      A     M   2002.5;
      =     L      0.0;
      BLD   103;
      A     I    367.3;
      =     L      0.1;
      BLD   103;
      A     I    367.4;
      =     L      0.2;
      BLD   103;
      A     I    367.6;
      =     L      0.4;
      BLD   103;
      A     I    367.7;
      =     L      0.6;
      BLD   103;
      A     I    368.0;
      =     L      1.0;
      BLD   103;
      A     I    368.1;
      =     L      1.2;
      BLD   103;
      A     M   2241.6;
      =     L      2.1;
      BLD   103;
      A     M   2241.7;
      =     L      2.2;
      BLD   103;
      AN    M   2004.0;
      AN    M   2004.1;
      AN    M   6060.1;
      AN    M   6460.0;
      AN    M   6480.0;
      AN    M   2004.2;
      A     M   2000.2;
      =     L      2.3;
      BLD   103;
      A(    ;
      O     I    150.1;
      O     I      0.1;
      )     ;
      =     L      2.5;
      BLD   103;
      A     M      0.5;
      =     L      2.6;
      BLD   103;
      CALL #S704_TL_DC_2ND_CLAMP2 (
           Enable_Aux               := L      0.0,
           Adv_Amount               := 1,
           Ret_Amount               := 5,
           LS_Adv1                  := L      0.1,
           LS_Ret1                  := L      0.2,
           LS_Ret2                  := L      0.4,
           LS_Ret3                  := L      0.6,
           LS_Ret4                  := L      1.0,
           LS_Ret5                  := L      1.2,
           SOL_Adv                  := L      2.1,
           SOL_Ret                  := L      2.2,
           M_Ready                  := L      2.3,
           T_CHK1                   := T#4S,
           T_CHK2                   := T#4S,
           PB_Error_Rst             := L      2.5,
           M_FLICK                  := L      2.6,
           M_Adv_Err                := M   2251.6,
           M_Ret_Err                := M   2251.7,
           Visu_Adv                 := DB51.DBW  748,
           Visu_Ret                 := DB51.DBW  750);
      NOP   0;
NETWORK
TITLE =
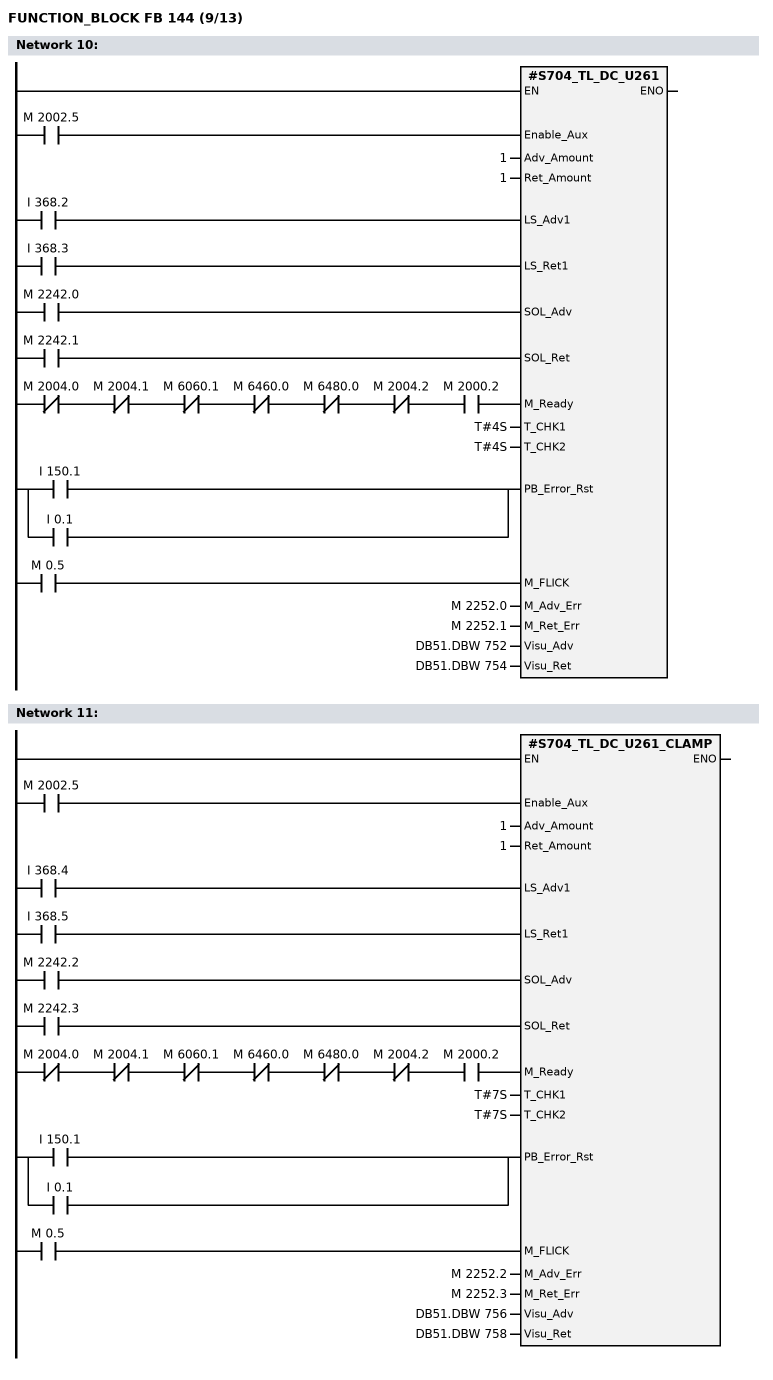

      A     M   2002.5;
      =     L      0.0;
      BLD   103;
      A     I    368.2;
      =     L      0.1;
      BLD   103;
      A     I    368.3;
      =     L      0.2;
      BLD   103;
      A     M   2242.0;
      =     L      2.1;
      BLD   103;
      A     M   2242.1;
      =     L      2.2;
      BLD   103;
      AN    M   2004.0;
      AN    M   2004.1;
      AN    M   6060.1;
      AN    M   6460.0;
      AN    M   6480.0;
      AN    M   2004.2;
      A     M   2000.2;
      =     L      2.3;
      BLD   103;
      A(    ;
      O     I    150.1;
      O     I      0.1;
      )     ;
      =     L      2.5;
      BLD   103;
      A     M      0.5;
      =     L      2.6;
      BLD   103;
      CALL #S704_TL_DC_U261 (
           Enable_Aux               := L      0.0,
           Adv_Amount               := 1,
           Ret_Amount               := 1,
           LS_Adv1                  := L      0.1,
           LS_Ret1                  := L      0.2,
           SOL_Adv                  := L      2.1,
           SOL_Ret                  := L      2.2,
           M_Ready                  := L      2.3,
           T_CHK1                   := T#4S,
           T_CHK2                   := T#4S,
           PB_Error_Rst             := L      2.5,
           M_FLICK                  := L      2.6,
           M_Adv_Err                := M   2252.0,
           M_Ret_Err                := M   2252.1,
           Visu_Adv                 := DB51.DBW  752,
           Visu_Ret                 := DB51.DBW  754);
      NOP   0;
NETWORK
TITLE =

      A     M   2002.5;
      =     L      0.0;
      BLD   103;
      A     I    368.4;
      =     L      0.1;
      BLD   103;
      A     I    368.5;
      =     L      0.2;
      BLD   103;
      A     M   2242.2;
      =     L      2.1;
      BLD   103;
      A     M   2242.3;
      =     L      2.2;
      BLD   103;
      AN    M   2004.0;
      AN    M   2004.1;
      AN    M   6060.1;
      AN    M   6460.0;
      AN    M   6480.0;
      AN    M   2004.2;
      A     M   2000.2;
      =     L      2.3;
      BLD   103;
      A(    ;
      O     I    150.1;
      O     I      0.1;
      )     ;
      =     L      2.5;
      BLD   103;
      A     M      0.5;
      =     L      2.6;
      BLD   103;
      CALL #S704_TL_DC_U261_CLAMP (
           Enable_Aux               := L      0.0,
           Adv_Amount               := 1,
           Ret_Amount               := 1,
           LS_Adv1                  := L      0.1,
           LS_Ret1                  := L      0.2,
           SOL_Adv                  := L      2.1,
           SOL_Ret                  := L      2.2,
           M_Ready                  := L      2.3,
           T_CHK1                   := T#7S,
           T_CHK2                   := T#7S,
           PB_Error_Rst             := L      2.5,
           M_FLICK                  := L      2.6,
           M_Adv_Err                := M   2252.2,
           M_Ret_Err                := M   2252.3,
           Visu_Adv                 := DB51.DBW  756,
           Visu_Ret                 := DB51.DBW  758);
      NOP   0;
NETWORK
TITLE =
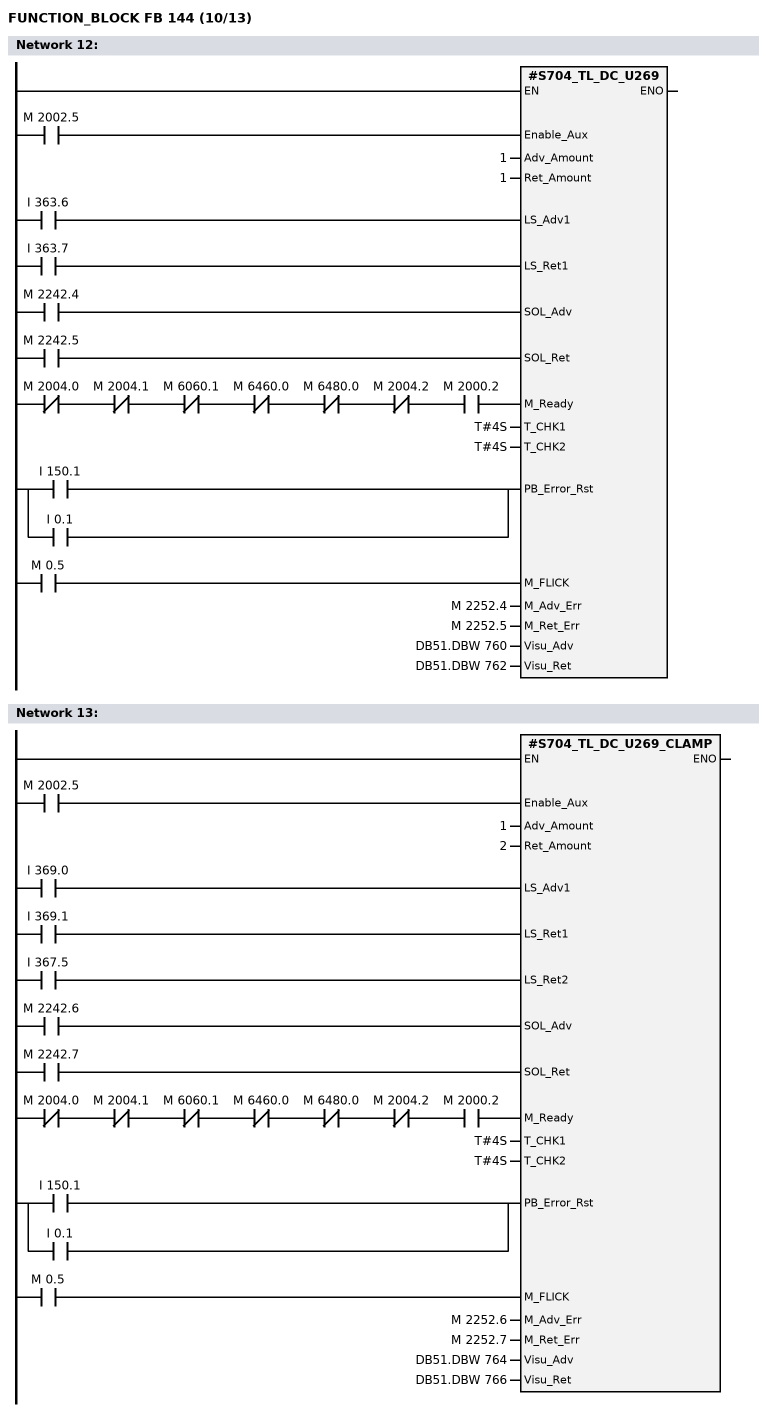

      A     M   2002.5;
      =     L      0.0;
      BLD   103;
      A     I    363.6;
      =     L      0.1;
      BLD   103;
      A     I    363.7;
      =     L      0.2;
      BLD   103;
      A     M   2242.4;
      =     L      2.1;
      BLD   103;
      A     M   2242.5;
      =     L      2.2;
      BLD   103;
      AN    M   2004.0;
      AN    M   2004.1;
      AN    M   6060.1;
      AN    M   6460.0;
      AN    M   6480.0;
      AN    M   2004.2;
      A     M   2000.2;
      =     L      2.3;
      BLD   103;
      A(    ;
      O     I    150.1;
      O     I      0.1;
      )     ;
      =     L      2.5;
      BLD   103;
      A     M      0.5;
      =     L      2.6;
      BLD   103;
      CALL #S704_TL_DC_U269 (
           Enable_Aux               := L      0.0,
           Adv_Amount               := 1,
           Ret_Amount               := 1,
           LS_Adv1                  := L      0.1,
           LS_Ret1                  := L      0.2,
           SOL_Adv                  := L      2.1,
           SOL_Ret                  := L      2.2,
           M_Ready                  := L      2.3,
           T_CHK1                   := T#4S,
           T_CHK2                   := T#4S,
           PB_Error_Rst             := L      2.5,
           M_FLICK                  := L      2.6,
           M_Adv_Err                := M   2252.4,
           M_Ret_Err                := M   2252.5,
           Visu_Adv                 := DB51.DBW  760,
           Visu_Ret                 := DB51.DBW  762);
      NOP   0;
NETWORK
TITLE =

      A     M   2002.5;
      =     L      0.0;
      BLD   103;
      A     I    369.0;
      =     L      0.1;
      BLD   103;
      A     I    369.1;
      =     L      0.2;
      BLD   103;
      A     I    367.5;
      =     L      0.4;
      BLD   103;
      A     M   2242.6;
      =     L      2.1;
      BLD   103;
      A     M   2242.7;
      =     L      2.2;
      BLD   103;
      AN    M   2004.0;
      AN    M   2004.1;
      AN    M   6060.1;
      AN    M   6460.0;
      AN    M   6480.0;
      AN    M   2004.2;
      A     M   2000.2;
      =     L      2.3;
      BLD   103;
      A(    ;
      O     I    150.1;
      O     I      0.1;
      )     ;
      =     L      2.5;
      BLD   103;
      A     M      0.5;
      =     L      2.6;
      BLD   103;
      CALL #S704_TL_DC_U269_CLAMP (
           Enable_Aux               := L      0.0,
           Adv_Amount               := 1,
           Ret_Amount               := 2,
           LS_Adv1                  := L      0.1,
           LS_Ret1                  := L      0.2,
           LS_Ret2                  := L      0.4,
           SOL_Adv                  := L      2.1,
           SOL_Ret                  := L      2.2,
           M_Ready                  := L      2.3,
           T_CHK1                   := T#4S,
           T_CHK2                   := T#4S,
           PB_Error_Rst             := L      2.5,
           M_FLICK                  := L      2.6,
           M_Adv_Err                := M   2252.6,
           M_Ret_Err                := M   2252.7,
           Visu_Adv                 := DB51.DBW  764,
           Visu_Ret                 := DB51.DBW  766);
      NOP   0;
NETWORK
TITLE =
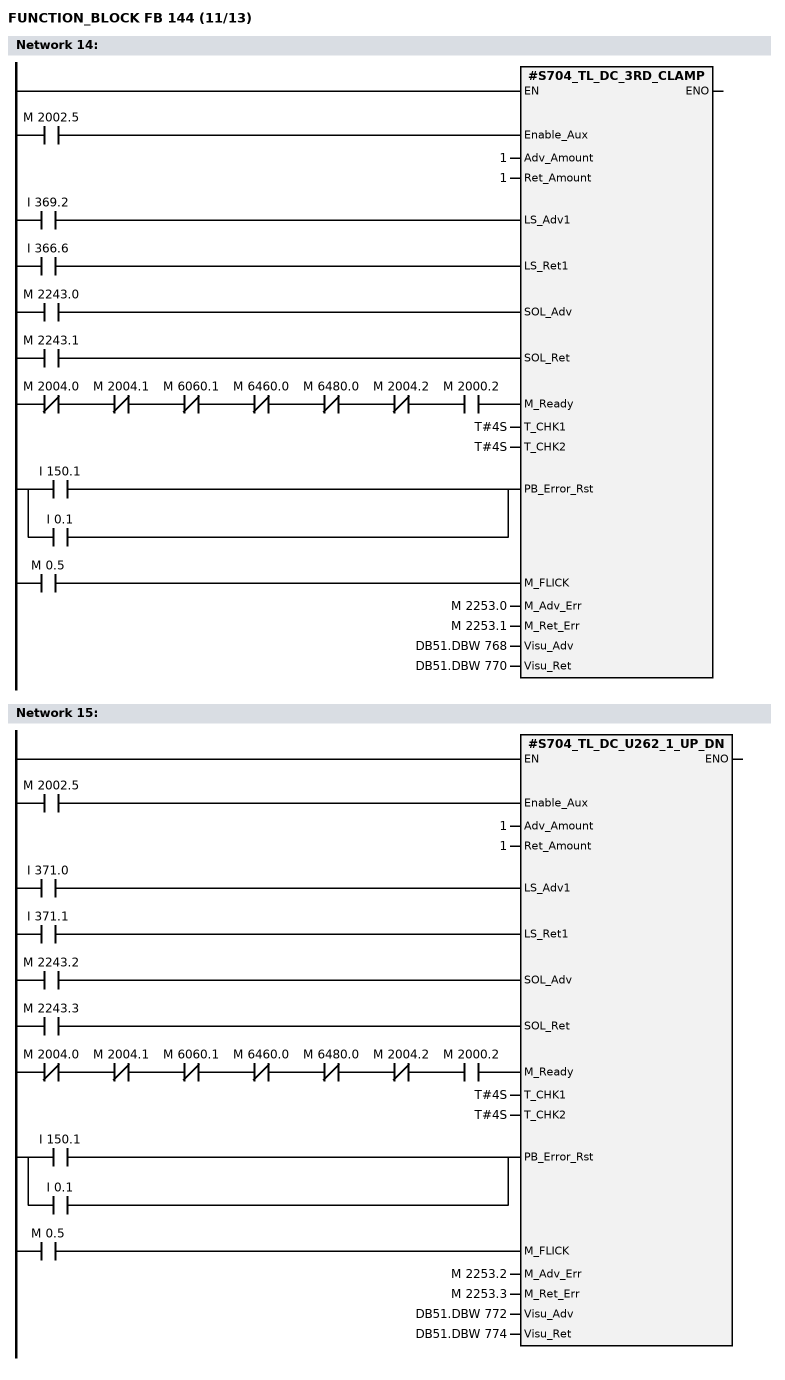

      A     M   2002.5;
      =     L      0.0;
      BLD   103;
      A     I    369.2;
      =     L      0.1;
      BLD   103;
      A     I    366.6;
      =     L      0.2;
      BLD   103;
      A     M   2243.0;
      =     L      2.1;
      BLD   103;
      A     M   2243.1;
      =     L      2.2;
      BLD   103;
      AN    M   2004.0;
      AN    M   2004.1;
      AN    M   6060.1;
      AN    M   6460.0;
      AN    M   6480.0;
      AN    M   2004.2;
      A     M   2000.2;
      =     L      2.3;
      BLD   103;
      A(    ;
      O     I    150.1;
      O     I      0.1;
      )     ;
      =     L      2.5;
      BLD   103;
      A     M      0.5;
      =     L      2.6;
      BLD   103;
      CALL #S704_TL_DC_3RD_CLAMP (
           Enable_Aux               := L      0.0,
           Adv_Amount               := 1,
           Ret_Amount               := 1,
           LS_Adv1                  := L      0.1,
           LS_Ret1                  := L      0.2,
           SOL_Adv                  := L      2.1,
           SOL_Ret                  := L      2.2,
           M_Ready                  := L      2.3,
           T_CHK1                   := T#4S,
           T_CHK2                   := T#4S,
           PB_Error_Rst             := L      2.5,
           M_FLICK                  := L      2.6,
           M_Adv_Err                := M   2253.0,
           M_Ret_Err                := M   2253.1,
           Visu_Adv                 := DB51.DBW  768,
           Visu_Ret                 := DB51.DBW  770);
      NOP   0;
NETWORK
TITLE =

      A     M   2002.5;
      =     L      0.0;
      BLD   103;
      A     I    371.0;
      =     L      0.1;
      BLD   103;
      A     I    371.1;
      =     L      0.2;
      BLD   103;
      A     M   2243.2;
      =     L      2.1;
      BLD   103;
      A     M   2243.3;
      =     L      2.2;
      BLD   103;
      AN    M   2004.0;
      AN    M   2004.1;
      AN    M   6060.1;
      AN    M   6460.0;
      AN    M   6480.0;
      AN    M   2004.2;
      A     M   2000.2;
      =     L      2.3;
      BLD   103;
      A(    ;
      O     I    150.1;
      O     I      0.1;
      )     ;
      =     L      2.5;
      BLD   103;
      A     M      0.5;
      =     L      2.6;
      BLD   103;
      CALL #S704_TL_DC_U262_1_UP_DN (
           Enable_Aux               := L      0.0,
           Adv_Amount               := 1,
           Ret_Amount               := 1,
           LS_Adv1                  := L      0.1,
           LS_Ret1                  := L      0.2,
           SOL_Adv                  := L      2.1,
           SOL_Ret                  := L      2.2,
           M_Ready                  := L      2.3,
           T_CHK1                   := T#4S,
           T_CHK2                   := T#4S,
           PB_Error_Rst             := L      2.5,
           M_FLICK                  := L      2.6,
           M_Adv_Err                := M   2253.2,
           M_Ret_Err                := M   2253.3,
           Visu_Adv                 := DB51.DBW  772,
           Visu_Ret                 := DB51.DBW  774);
      NOP   0;
NETWORK
TITLE =
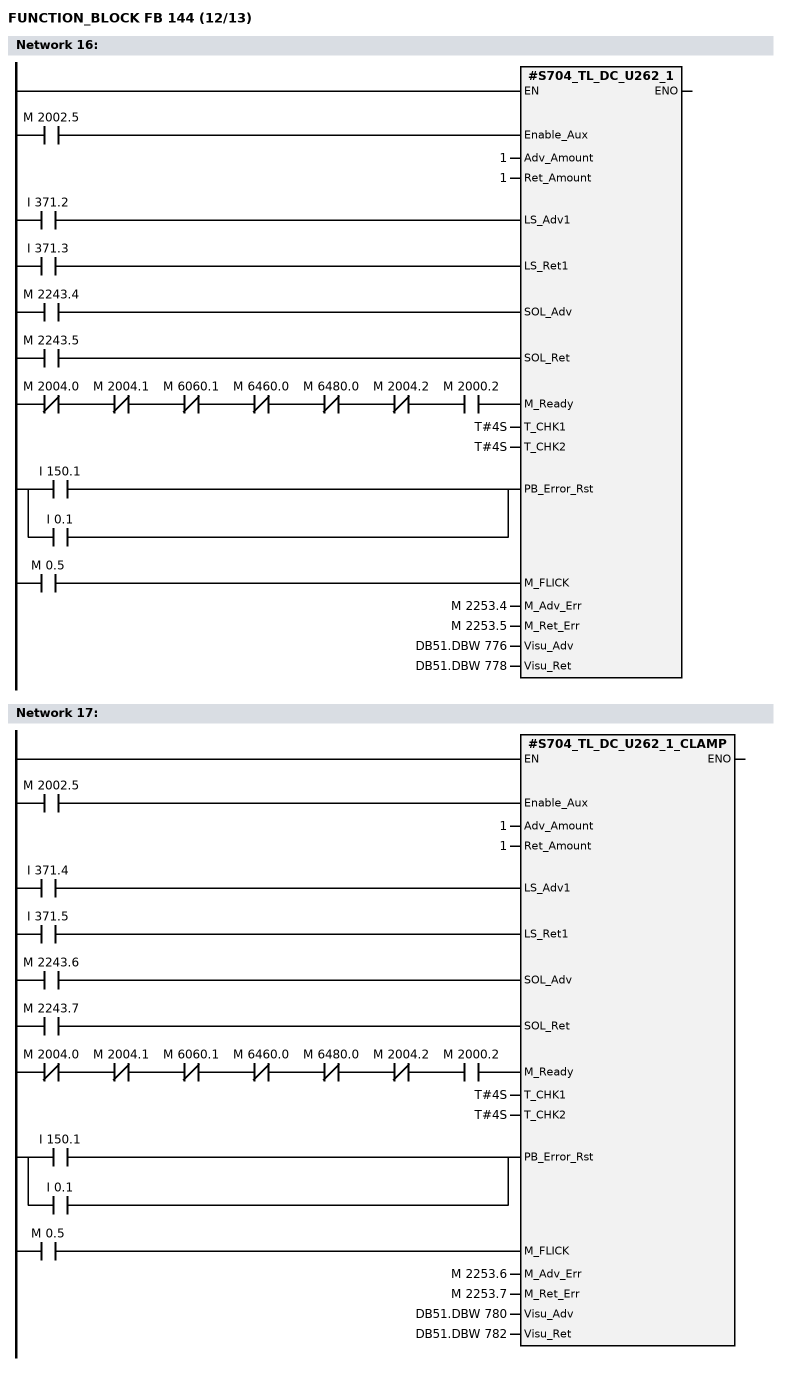

      A     M   2002.5;
      =     L      0.0;
      BLD   103;
      A     I    371.2;
      =     L      0.1;
      BLD   103;
      A     I    371.3;
      =     L      0.2;
      BLD   103;
      A     M   2243.4;
      =     L      2.1;
      BLD   103;
      A     M   2243.5;
      =     L      2.2;
      BLD   103;
      AN    M   2004.0;
      AN    M   2004.1;
      AN    M   6060.1;
      AN    M   6460.0;
      AN    M   6480.0;
      AN    M   2004.2;
      A     M   2000.2;
      =     L      2.3;
      BLD   103;
      A(    ;
      O     I    150.1;
      O     I      0.1;
      )     ;
      =     L      2.5;
      BLD   103;
      A     M      0.5;
      =     L      2.6;
      BLD   103;
      CALL #S704_TL_DC_U262_1 (
           Enable_Aux               := L      0.0,
           Adv_Amount               := 1,
           Ret_Amount               := 1,
           LS_Adv1                  := L      0.1,
           LS_Ret1                  := L      0.2,
           SOL_Adv                  := L      2.1,
           SOL_Ret                  := L      2.2,
           M_Ready                  := L      2.3,
           T_CHK1                   := T#4S,
           T_CHK2                   := T#4S,
           PB_Error_Rst             := L      2.5,
           M_FLICK                  := L      2.6,
           M_Adv_Err                := M   2253.4,
           M_Ret_Err                := M   2253.5,
           Visu_Adv                 := DB51.DBW  776,
           Visu_Ret                 := DB51.DBW  778);
      NOP   0;
NETWORK
TITLE =

      A     M   2002.5;
      =     L      0.0;
      BLD   103;
      A     I    371.4;
      =     L      0.1;
      BLD   103;
      A     I    371.5;
      =     L      0.2;
      BLD   103;
      A     M   2243.6;
      =     L      2.1;
      BLD   103;
      A     M   2243.7;
      =     L      2.2;
      BLD   103;
      AN    M   2004.0;
      AN    M   2004.1;
      AN    M   6060.1;
      AN    M   6460.0;
      AN    M   6480.0;
      AN    M   2004.2;
      A     M   2000.2;
      =     L      2.3;
      BLD   103;
      A(    ;
      O     I    150.1;
      O     I      0.1;
      )     ;
      =     L      2.5;
      BLD   103;
      A     M      0.5;
      =     L      2.6;
      BLD   103;
      CALL #S704_TL_DC_U262_1_CLAMP (
           Enable_Aux               := L      0.0,
           Adv_Amount               := 1,
           Ret_Amount               := 1,
           LS_Adv1                  := L      0.1,
           LS_Ret1                  := L      0.2,
           SOL_Adv                  := L      2.1,
           SOL_Ret                  := L      2.2,
           M_Ready                  := L      2.3,
           T_CHK1                   := T#4S,
           T_CHK2                   := T#4S,
           PB_Error_Rst             := L      2.5,
           M_FLICK                  := L      2.6,
           M_Adv_Err                := M   2253.6,
           M_Ret_Err                := M   2253.7,
           Visu_Adv                 := DB51.DBW  780,
           Visu_Ret                 := DB51.DBW  782);
      NOP   0;
NETWORK
TITLE =
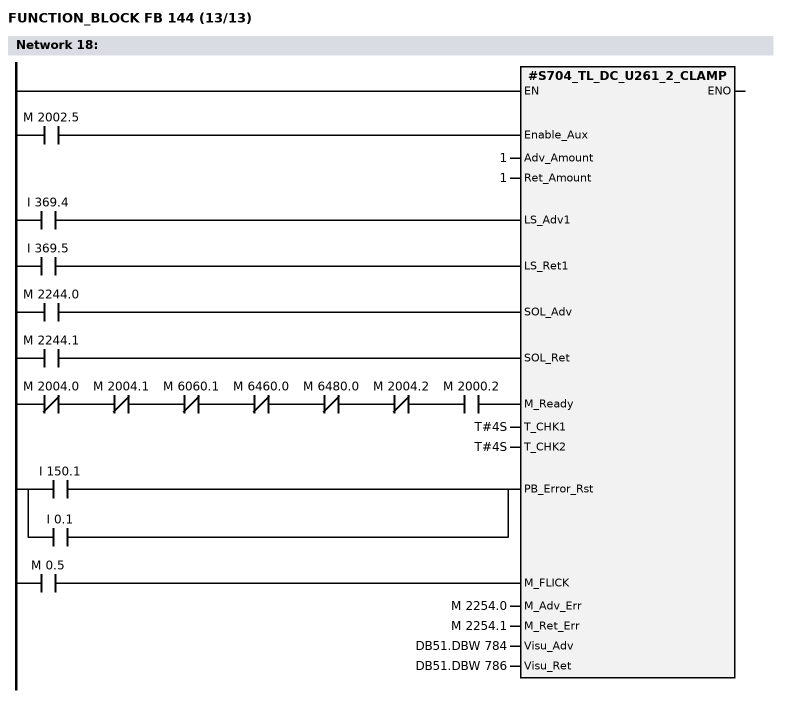

      A     M   2002.5;
      =     L      0.0;
      BLD   103;
      A     I    369.4;
      =     L      0.1;
      BLD   103;
      A     I    369.5;
      =     L      0.2;
      BLD   103;
      A     M   2244.0;
      =     L      2.1;
      BLD   103;
      A     M   2244.1;
      =     L      2.2;
      BLD   103;
      AN    M   2004.0;
      AN    M   2004.1;
      AN    M   6060.1;
      AN    M   6460.0;
      AN    M   6480.0;
      AN    M   2004.2;
      A     M   2000.2;
      =     L      2.3;
      BLD   103;
      A(    ;
      O     I    150.1;
      O     I      0.1;
      )     ;
      =     L      2.5;
      BLD   103;
      A     M      0.5;
      =     L      2.6;
      BLD   103;
      CALL #S704_TL_DC_U261_2_CLAMP (
           Enable_Aux               := L      0.0,
           Adv_Amount               := 1,
           Ret_Amount               := 1,
           LS_Adv1                  := L      0.1,
           LS_Ret1                  := L      0.2,
           SOL_Adv                  := L      2.1,
           SOL_Ret                  := L      2.2,
           M_Ready                  := L      2.3,
           T_CHK1                   := T#4S,
           T_CHK2                   := T#4S,
           PB_Error_Rst             := L      2.5,
           M_FLICK                  := L      2.6,
           M_Adv_Err                := M   2254.0,
           M_Ret_Err                := M   2254.1,
           Visu_Adv                 := DB51.DBW  784,
           Visu_Ret                 := DB51.DBW  786);
      NOP   0;
END_FUNCTION_BLOCK

DATA_BLOCK DB 144
TITLE =
VERSION : 0.0

 FB 144
BEGIN
   S704_TL_DC_PIN.Enable_Aux := FALSE;
   S704_TL_DC_PIN.Adv_Amount := 0;
   S704_TL_DC_PIN.Ret_Amount := 0;
   S704_TL_DC_PIN.LS_Adv1 := FALSE;
   S704_TL_DC_PIN.LS_Ret1 := FALSE;
   S704_TL_DC_PIN.LS_Adv2 := FALSE;
   S704_TL_DC_PIN.LS_Ret2 := FALSE;
   S704_TL_DC_PIN.LS_Adv3 := FALSE;
   S704_TL_DC_PIN.LS_Ret3 := FALSE;
   S704_TL_DC_PIN.LS_Adv4 := FALSE;
   S704_TL_DC_PIN.LS_Ret4 := FALSE;
   S704_TL_DC_PIN.LS_Adv5 := FALSE;
   S704_TL_DC_PIN.LS_Ret5 := FALSE;
   S704_TL_DC_PIN.LS_Adv6 := FALSE;
   S704_TL_DC_PIN.LS_Ret6 := FALSE;
   S704_TL_DC_PIN.LS_Adv7 := FALSE;
   S704_TL_DC_PIN.LS_Ret7 := FALSE;
   S704_TL_DC_PIN.LS_Adv8 := FALSE;
   S704_TL_DC_PIN.LS_Ret8 := FALSE;
   S704_TL_DC_PIN.SOL_Adv := FALSE;
   S704_TL_DC_PIN.SOL_Ret := FALSE;
   S704_TL_DC_PIN.M_Ready := FALSE;
   S704_TL_DC_PIN.T_CHK1 := T#0MS;
   S704_TL_DC_PIN.T_CHK2 := T#0MS;
   S704_TL_DC_PIN.PB_Lamp_CHK := FALSE;
   S704_TL_DC_PIN.PB_Error_Rst := FALSE;
   S704_TL_DC_PIN.M_FLICK := FALSE;
   S704_TL_DC_PIN.M_Adv_Err := FALSE;
   S704_TL_DC_PIN.M_Ret_Err := FALSE;
   S704_TL_DC_PIN.LP_Adv := FALSE;
   S704_TL_DC_PIN.LP_Ret := FALSE;
   S704_TL_DC_PIN.Visu_Adv := W#16#0;
   S704_TL_DC_PIN.Visu_Ret := W#16#0;
   S704_TL_DC_PIN.Error_T1.IN := FALSE;
   S704_TL_DC_PIN.Error_T1.PT := T#0MS;
   S704_TL_DC_PIN.Error_T1.Q := FALSE;
   S704_TL_DC_PIN.Error_T1.ET := T#0MS;
   S704_TL_DC_PIN.Error_T1.STATE := B#16#0;
   S704_TL_DC_PIN.Error_T1.STIME := T#0MS;
   S704_TL_DC_PIN.Error_T1.ATIME := T#0MS;
   S704_TL_DC_PIN.Error_T2.IN := FALSE;
   S704_TL_DC_PIN.Error_T2.PT := T#0MS;
   S704_TL_DC_PIN.Error_T2.Q := FALSE;
   S704_TL_DC_PIN.Error_T2.ET := T#0MS;
   S704_TL_DC_PIN.Error_T2.STATE := B#16#0;
   S704_TL_DC_PIN.Error_T2.STIME := T#0MS;
   S704_TL_DC_PIN.Error_T2.ATIME := T#0MS;
   S704_TL_DC_PIN.Adv_End_Aux := FALSE;
   S704_TL_DC_PIN.Ret_End_Aux := FALSE;
   S704_TL_DC_PIN.CHK_Aux1 := FALSE;
   S704_TL_DC_PIN.CHK_Aux2 := FALSE;
   S704_TL_DC_PIN.Error_T1_DN := FALSE;
   S704_TL_DC_PIN.Error_T2_DN := FALSE;
   S704_TL_DC_PIN.Adv_Memo := FALSE;
   S704_TL_DC_PIN.Visu_Adv_Arr[0] := FALSE;
   S704_TL_DC_PIN.Visu_Adv_Arr[1] := FALSE;
   S704_TL_DC_PIN.Visu_Adv_Arr[2] := FALSE;
   S704_TL_DC_PIN.Visu_Adv_Arr[3] := FALSE;
   S704_TL_DC_PIN.Visu_Adv_Arr[4] := FALSE;
   S704_TL_DC_PIN.Visu_Adv_Arr[5] := FALSE;
   S704_TL_DC_PIN.Visu_Adv_Arr[6] := FALSE;
   S704_TL_DC_PIN.Visu_Adv_Arr[7] := FALSE;
   S704_TL_DC_PIN.Visu_Adv_Arr[8] := FALSE;
   S704_TL_DC_PIN.Visu_Adv_Arr[9] := FALSE;
   S704_TL_DC_PIN.Visu_Adv_Arr[10] := FALSE;
   S704_TL_DC_PIN.Visu_Adv_Arr[11] := FALSE;
   S704_TL_DC_PIN.Visu_Adv_Arr[12] := FALSE;
   S704_TL_DC_PIN.Visu_Adv_Arr[13] := FALSE;
   S704_TL_DC_PIN.Visu_Adv_Arr[14] := FALSE;
   S704_TL_DC_PIN.Visu_Adv_Arr[15] := FALSE;
   S704_TL_DC_PIN.Visu_Ret_Arr[0] := FALSE;
   S704_TL_DC_PIN.Visu_Ret_Arr[1] := FALSE;
   S704_TL_DC_PIN.Visu_Ret_Arr[2] := FALSE;
   S704_TL_DC_PIN.Visu_Ret_Arr[3] := FALSE;
   S704_TL_DC_PIN.Visu_Ret_Arr[4] := FALSE;
   S704_TL_DC_PIN.Visu_Ret_Arr[5] := FALSE;
   S704_TL_DC_PIN.Visu_Ret_Arr[6] := FALSE;
   S704_TL_DC_PIN.Visu_Ret_Arr[7] := FALSE;
   S704_TL_DC_PIN.Visu_Ret_Arr[8] := FALSE;
   S704_TL_DC_PIN.Visu_Ret_Arr[9] := FALSE;
   S704_TL_DC_PIN.Visu_Ret_Arr[10] := FALSE;
   S704_TL_DC_PIN.Visu_Ret_Arr[11] := FALSE;
   S704_TL_DC_PIN.Visu_Ret_Arr[12] := FALSE;
   S704_TL_DC_PIN.Visu_Ret_Arr[13] := FALSE;
   S704_TL_DC_PIN.Visu_Ret_Arr[14] := FALSE;
   S704_TL_DC_PIN.Visu_Ret_Arr[15] := FALSE;
   S704_TL_DC_PIN.BLK_Move_Ret := 0;
   S704_TL_DC_PIN.Enable := FALSE;
   S704_TL_DC_PIN.Adv_End := FALSE;
   S704_TL_DC_PIN.Ret_End := FALSE;
   S704_TL_DC_LATCH1.Enable_Aux := FALSE;
   S704_TL_DC_LATCH1.Adv_Amount := 0;
   S704_TL_DC_LATCH1.Ret_Amount := 0;
   S704_TL_DC_LATCH1.LS_Adv1 := FALSE;
   S704_TL_DC_LATCH1.LS_Ret1 := FALSE;
   S704_TL_DC_LATCH1.LS_Adv2 := FALSE;
   S704_TL_DC_LATCH1.LS_Ret2 := FALSE;
   S704_TL_DC_LATCH1.LS_Adv3 := FALSE;
   S704_TL_DC_LATCH1.LS_Ret3 := FALSE;
   S704_TL_DC_LATCH1.LS_Adv4 := FALSE;
   S704_TL_DC_LATCH1.LS_Ret4 := FALSE;
   S704_TL_DC_LATCH1.LS_Adv5 := FALSE;
   S704_TL_DC_LATCH1.LS_Ret5 := FALSE;
   S704_TL_DC_LATCH1.LS_Adv6 := FALSE;
   S704_TL_DC_LATCH1.LS_Ret6 := FALSE;
   S704_TL_DC_LATCH1.LS_Adv7 := FALSE;
   S704_TL_DC_LATCH1.LS_Ret7 := FALSE;
   S704_TL_DC_LATCH1.LS_Adv8 := FALSE;
   S704_TL_DC_LATCH1.LS_Ret8 := FALSE;
   S704_TL_DC_LATCH1.SOL_Adv := FALSE;
   S704_TL_DC_LATCH1.SOL_Ret := FALSE;
   S704_TL_DC_LATCH1.M_Ready := FALSE;
   S704_TL_DC_LATCH1.T_CHK1 := T#0MS;
   S704_TL_DC_LATCH1.T_CHK2 := T#0MS;
   S704_TL_DC_LATCH1.PB_Lamp_CHK := FALSE;
   S704_TL_DC_LATCH1.PB_Error_Rst := FALSE;
   S704_TL_DC_LATCH1.M_FLICK := FALSE;
   S704_TL_DC_LATCH1.M_Adv_Err := FALSE;
   S704_TL_DC_LATCH1.M_Ret_Err := FALSE;
   S704_TL_DC_LATCH1.LP_Adv := FALSE;
   S704_TL_DC_LATCH1.LP_Ret := FALSE;
   S704_TL_DC_LATCH1.Visu_Adv := W#16#0;
   S704_TL_DC_LATCH1.Visu_Ret := W#16#0;
   S704_TL_DC_LATCH1.Error_T1.IN := FALSE;
   S704_TL_DC_LATCH1.Error_T1.PT := T#0MS;
   S704_TL_DC_LATCH1.Error_T1.Q := FALSE;
   S704_TL_DC_LATCH1.Error_T1.ET := T#0MS;
   S704_TL_DC_LATCH1.Error_T1.STATE := B#16#0;
   S704_TL_DC_LATCH1.Error_T1.STIME := T#0MS;
   S704_TL_DC_LATCH1.Error_T1.ATIME := T#0MS;
   S704_TL_DC_LATCH1.Error_T2.IN := FALSE;
   S704_TL_DC_LATCH1.Error_T2.PT := T#0MS;
   S704_TL_DC_LATCH1.Error_T2.Q := FALSE;
   S704_TL_DC_LATCH1.Error_T2.ET := T#0MS;
   S704_TL_DC_LATCH1.Error_T2.STATE := B#16#0;
   S704_TL_DC_LATCH1.Error_T2.STIME := T#0MS;
   S704_TL_DC_LATCH1.Error_T2.ATIME := T#0MS;
   S704_TL_DC_LATCH1.Adv_End_Aux := FALSE;
   S704_TL_DC_LATCH1.Ret_End_Aux := FALSE;
   S704_TL_DC_LATCH1.CHK_Aux1 := FALSE;
   S704_TL_DC_LATCH1.CHK_Aux2 := FALSE;
   S704_TL_DC_LATCH1.Error_T1_DN := FALSE;
   S704_TL_DC_LATCH1.Error_T2_DN := FALSE;
   S704_TL_DC_LATCH1.Adv_Memo := FALSE;
   S704_TL_DC_LATCH1.Visu_Adv_Arr[0] := FALSE;
   S704_TL_DC_LATCH1.Visu_Adv_Arr[1] := FALSE;
   S704_TL_DC_LATCH1.Visu_Adv_Arr[2] := FALSE;
   S704_TL_DC_LATCH1.Visu_Adv_Arr[3] := FALSE;
   S704_TL_DC_LATCH1.Visu_Adv_Arr[4] := FALSE;
   S704_TL_DC_LATCH1.Visu_Adv_Arr[5] := FALSE;
   S704_TL_DC_LATCH1.Visu_Adv_Arr[6] := FALSE;
   S704_TL_DC_LATCH1.Visu_Adv_Arr[7] := FALSE;
   S704_TL_DC_LATCH1.Visu_Adv_Arr[8] := FALSE;
   S704_TL_DC_LATCH1.Visu_Adv_Arr[9] := FALSE;
   S704_TL_DC_LATCH1.Visu_Adv_Arr[10] := FALSE;
   S704_TL_DC_LATCH1.Visu_Adv_Arr[11] := FALSE;
   S704_TL_DC_LATCH1.Visu_Adv_Arr[12] := FALSE;
   S704_TL_DC_LATCH1.Visu_Adv_Arr[13] := FALSE;
   S704_TL_DC_LATCH1.Visu_Adv_Arr[14] := FALSE;
   S704_TL_DC_LATCH1.Visu_Adv_Arr[15] := FALSE;
   S704_TL_DC_LATCH1.Visu_Ret_Arr[0] := FALSE;
   S704_TL_DC_LATCH1.Visu_Ret_Arr[1] := FALSE;
   S704_TL_DC_LATCH1.Visu_Ret_Arr[2] := FALSE;
   S704_TL_DC_LATCH1.Visu_Ret_Arr[3] := FALSE;
   S704_TL_DC_LATCH1.Visu_Ret_Arr[4] := FALSE;
   S704_TL_DC_LATCH1.Visu_Ret_Arr[5] := FALSE;
   S704_TL_DC_LATCH1.Visu_Ret_Arr[6] := FALSE;
   S704_TL_DC_LATCH1.Visu_Ret_Arr[7] := FALSE;
   S704_TL_DC_LATCH1.Visu_Ret_Arr[8] := FALSE;
   S704_TL_DC_LATCH1.Visu_Ret_Arr[9] := FALSE;
   S704_TL_DC_LATCH1.Visu_Ret_Arr[10] := FALSE;
   S704_TL_DC_LATCH1.Visu_Ret_Arr[11] := FALSE;
   S704_TL_DC_LATCH1.Visu_Ret_Arr[12] := FALSE;
   S704_TL_DC_LATCH1.Visu_Ret_Arr[13] := FALSE;
   S704_TL_DC_LATCH1.Visu_Ret_Arr[14] := FALSE;
   S704_TL_DC_LATCH1.Visu_Ret_Arr[15] := FALSE;
   S704_TL_DC_LATCH1.BLK_Move_Ret := 0;
   S704_TL_DC_LATCH1.Enable := FALSE;
   S704_TL_DC_LATCH1.Adv_End := FALSE;
   S704_TL_DC_LATCH1.Ret_End := FALSE;
   S704_TL_DC_LATCH2.Enable_Aux := FALSE;
   S704_TL_DC_LATCH2.Adv_Amount := 0;
   S704_TL_DC_LATCH2.Ret_Amount := 0;
   S704_TL_DC_LATCH2.LS_Adv1 := FALSE;
   S704_TL_DC_LATCH2.LS_Ret1 := FALSE;
   S704_TL_DC_LATCH2.LS_Adv2 := FALSE;
   S704_TL_DC_LATCH2.LS_Ret2 := FALSE;
   S704_TL_DC_LATCH2.LS_Adv3 := FALSE;
   S704_TL_DC_LATCH2.LS_Ret3 := FALSE;
   S704_TL_DC_LATCH2.LS_Adv4 := FALSE;
   S704_TL_DC_LATCH2.LS_Ret4 := FALSE;
   S704_TL_DC_LATCH2.LS_Adv5 := FALSE;
   S704_TL_DC_LATCH2.LS_Ret5 := FALSE;
   S704_TL_DC_LATCH2.LS_Adv6 := FALSE;
   S704_TL_DC_LATCH2.LS_Ret6 := FALSE;
   S704_TL_DC_LATCH2.LS_Adv7 := FALSE;
   S704_TL_DC_LATCH2.LS_Ret7 := FALSE;
   S704_TL_DC_LATCH2.LS_Adv8 := FALSE;
   S704_TL_DC_LATCH2.LS_Ret8 := FALSE;
   S704_TL_DC_LATCH2.SOL_Adv := FALSE;
   S704_TL_DC_LATCH2.SOL_Ret := FALSE;
   S704_TL_DC_LATCH2.M_Ready := FALSE;
   S704_TL_DC_LATCH2.T_CHK1 := T#0MS;
   S704_TL_DC_LATCH2.T_CHK2 := T#0MS;
   S704_TL_DC_LATCH2.PB_Lamp_CHK := FALSE;
   S704_TL_DC_LATCH2.PB_Error_Rst := FALSE;
   S704_TL_DC_LATCH2.M_FLICK := FALSE;
   S704_TL_DC_LATCH2.M_Adv_Err := FALSE;
   S704_TL_DC_LATCH2.M_Ret_Err := FALSE;
   S704_TL_DC_LATCH2.LP_Adv := FALSE;
   S704_TL_DC_LATCH2.LP_Ret := FALSE;
   S704_TL_DC_LATCH2.Visu_Adv := W#16#0;
   S704_TL_DC_LATCH2.Visu_Ret := W#16#0;
   S704_TL_DC_LATCH2.Error_T1.IN := FALSE;
   S704_TL_DC_LATCH2.Error_T1.PT := T#0MS;
   S704_TL_DC_LATCH2.Error_T1.Q := FALSE;
   S704_TL_DC_LATCH2.Error_T1.ET := T#0MS;
   S704_TL_DC_LATCH2.Error_T1.STATE := B#16#0;
   S704_TL_DC_LATCH2.Error_T1.STIME := T#0MS;
   S704_TL_DC_LATCH2.Error_T1.ATIME := T#0MS;
   S704_TL_DC_LATCH2.Error_T2.IN := FALSE;
   S704_TL_DC_LATCH2.Error_T2.PT := T#0MS;
   S704_TL_DC_LATCH2.Error_T2.Q := FALSE;
   S704_TL_DC_LATCH2.Error_T2.ET := T#0MS;
   S704_TL_DC_LATCH2.Error_T2.STATE := B#16#0;
   S704_TL_DC_LATCH2.Error_T2.STIME := T#0MS;
   S704_TL_DC_LATCH2.Error_T2.ATIME := T#0MS;
   S704_TL_DC_LATCH2.Adv_End_Aux := FALSE;
   S704_TL_DC_LATCH2.Ret_End_Aux := FALSE;
   S704_TL_DC_LATCH2.CHK_Aux1 := FALSE;
   S704_TL_DC_LATCH2.CHK_Aux2 := FALSE;
   S704_TL_DC_LATCH2.Error_T1_DN := FALSE;
   S704_TL_DC_LATCH2.Error_T2_DN := FALSE;
   S704_TL_DC_LATCH2.Adv_Memo := FALSE;
   S704_TL_DC_LATCH2.Visu_Adv_Arr[0] := FALSE;
   S704_TL_DC_LATCH2.Visu_Adv_Arr[1] := FALSE;
   S704_TL_DC_LATCH2.Visu_Adv_Arr[2] := FALSE;
   S704_TL_DC_LATCH2.Visu_Adv_Arr[3] := FALSE;
   S704_TL_DC_LATCH2.Visu_Adv_Arr[4] := FALSE;
   S704_TL_DC_LATCH2.Visu_Adv_Arr[5] := FALSE;
   S704_TL_DC_LATCH2.Visu_Adv_Arr[6] := FALSE;
   S704_TL_DC_LATCH2.Visu_Adv_Arr[7] := FALSE;
   S704_TL_DC_LATCH2.Visu_Adv_Arr[8] := FALSE;
   S704_TL_DC_LATCH2.Visu_Adv_Arr[9] := FALSE;
   S704_TL_DC_LATCH2.Visu_Adv_Arr[10] := FALSE;
   S704_TL_DC_LATCH2.Visu_Adv_Arr[11] := FALSE;
   S704_TL_DC_LATCH2.Visu_Adv_Arr[12] := FALSE;
   S704_TL_DC_LATCH2.Visu_Adv_Arr[13] := FALSE;
   S704_TL_DC_LATCH2.Visu_Adv_Arr[14] := FALSE;
   S704_TL_DC_LATCH2.Visu_Adv_Arr[15] := FALSE;
   S704_TL_DC_LATCH2.Visu_Ret_Arr[0] := FALSE;
   S704_TL_DC_LATCH2.Visu_Ret_Arr[1] := FALSE;
   S704_TL_DC_LATCH2.Visu_Ret_Arr[2] := FALSE;
   S704_TL_DC_LATCH2.Visu_Ret_Arr[3] := FALSE;
   S704_TL_DC_LATCH2.Visu_Ret_Arr[4] := FALSE;
   S704_TL_DC_LATCH2.Visu_Ret_Arr[5] := FALSE;
   S704_TL_DC_LATCH2.Visu_Ret_Arr[6] := FALSE;
   S704_TL_DC_LATCH2.Visu_Ret_Arr[7] := FALSE;
   S704_TL_DC_LATCH2.Visu_Ret_Arr[8] := FALSE;
   S704_TL_DC_LATCH2.Visu_Ret_Arr[9] := FALSE;
   S704_TL_DC_LATCH2.Visu_Ret_Arr[10] := FALSE;
   S704_TL_DC_LATCH2.Visu_Ret_Arr[11] := FALSE;
   S704_TL_DC_LATCH2.Visu_Ret_Arr[12] := FALSE;
   S704_TL_DC_LATCH2.Visu_Ret_Arr[13] := FALSE;
   S704_TL_DC_LATCH2.Visu_Ret_Arr[14] := FALSE;
   S704_TL_DC_LATCH2.Visu_Ret_Arr[15] := FALSE;
   S704_TL_DC_LATCH2.BLK_Move_Ret := 0;
   S704_TL_DC_LATCH2.Enable := FALSE;
   S704_TL_DC_LATCH2.Adv_End := FALSE;
   S704_TL_DC_LATCH2.Ret_End := FALSE;
   S704_TL_DC_1ST_CLAMP1.Enable_Aux := FALSE;
   S704_TL_DC_1ST_CLAMP1.Adv_Amount := 0;
   S704_TL_DC_1ST_CLAMP1.Ret_Amount := 0;
   S704_TL_DC_1ST_CLAMP1.LS_Adv1 := FALSE;
   S704_TL_DC_1ST_CLAMP1.LS_Ret1 := FALSE;
   S704_TL_DC_1ST_CLAMP1.LS_Adv2 := FALSE;
   S704_TL_DC_1ST_CLAMP1.LS_Ret2 := FALSE;
   S704_TL_DC_1ST_CLAMP1.LS_Adv3 := FALSE;
   S704_TL_DC_1ST_CLAMP1.LS_Ret3 := FALSE;
   S704_TL_DC_1ST_CLAMP1.LS_Adv4 := FALSE;
   S704_TL_DC_1ST_CLAMP1.LS_Ret4 := FALSE;
   S704_TL_DC_1ST_CLAMP1.LS_Adv5 := FALSE;
   S704_TL_DC_1ST_CLAMP1.LS_Ret5 := FALSE;
   S704_TL_DC_1ST_CLAMP1.LS_Adv6 := FALSE;
   S704_TL_DC_1ST_CLAMP1.LS_Ret6 := FALSE;
   S704_TL_DC_1ST_CLAMP1.LS_Adv7 := FALSE;
   S704_TL_DC_1ST_CLAMP1.LS_Ret7 := FALSE;
   S704_TL_DC_1ST_CLAMP1.LS_Adv8 := FALSE;
   S704_TL_DC_1ST_CLAMP1.LS_Ret8 := FALSE;
   S704_TL_DC_1ST_CLAMP1.SOL_Adv := FALSE;
   S704_TL_DC_1ST_CLAMP1.SOL_Ret := FALSE;
   S704_TL_DC_1ST_CLAMP1.M_Ready := FALSE;
   S704_TL_DC_1ST_CLAMP1.T_CHK1 := T#0MS;
   S704_TL_DC_1ST_CLAMP1.T_CHK2 := T#0MS;
   S704_TL_DC_1ST_CLAMP1.PB_Lamp_CHK := FALSE;
   S704_TL_DC_1ST_CLAMP1.PB_Error_Rst := FALSE;
   S704_TL_DC_1ST_CLAMP1.M_FLICK := FALSE;
   S704_TL_DC_1ST_CLAMP1.M_Adv_Err := FALSE;
   S704_TL_DC_1ST_CLAMP1.M_Ret_Err := FALSE;
   S704_TL_DC_1ST_CLAMP1.LP_Adv := FALSE;
   S704_TL_DC_1ST_CLAMP1.LP_Ret := FALSE;
   S704_TL_DC_1ST_CLAMP1.Visu_Adv := W#16#0;
   S704_TL_DC_1ST_CLAMP1.Visu_Ret := W#16#0;
   S704_TL_DC_1ST_CLAMP1.Error_T1.IN := FALSE;
   S704_TL_DC_1ST_CLAMP1.Error_T1.PT := T#0MS;
   S704_TL_DC_1ST_CLAMP1.Error_T1.Q := FALSE;
   S704_TL_DC_1ST_CLAMP1.Error_T1.ET := T#0MS;
   S704_TL_DC_1ST_CLAMP1.Error_T1.STATE := B#16#0;
   S704_TL_DC_1ST_CLAMP1.Error_T1.STIME := T#0MS;
   S704_TL_DC_1ST_CLAMP1.Error_T1.ATIME := T#0MS;
   S704_TL_DC_1ST_CLAMP1.Error_T2.IN := FALSE;
   S704_TL_DC_1ST_CLAMP1.Error_T2.PT := T#0MS;
   S704_TL_DC_1ST_CLAMP1.Error_T2.Q := FALSE;
   S704_TL_DC_1ST_CLAMP1.Error_T2.ET := T#0MS;
   S704_TL_DC_1ST_CLAMP1.Error_T2.STATE := B#16#0;
   S704_TL_DC_1ST_CLAMP1.Error_T2.STIME := T#0MS;
   S704_TL_DC_1ST_CLAMP1.Error_T2.ATIME := T#0MS;
   S704_TL_DC_1ST_CLAMP1.Adv_End_Aux := FALSE;
   S704_TL_DC_1ST_CLAMP1.Ret_End_Aux := FALSE;
   S704_TL_DC_1ST_CLAMP1.CHK_Aux1 := FALSE;
   S704_TL_DC_1ST_CLAMP1.CHK_Aux2 := FALSE;
   S704_TL_DC_1ST_CLAMP1.Error_T1_DN := FALSE;
   S704_TL_DC_1ST_CLAMP1.Error_T2_DN := FALSE;
   S704_TL_DC_1ST_CLAMP1.Adv_Memo := FALSE;
   S704_TL_DC_1ST_CLAMP1.Visu_Adv_Arr[0] := FALSE;
   S704_TL_DC_1ST_CLAMP1.Visu_Adv_Arr[1] := FALSE;
   S704_TL_DC_1ST_CLAMP1.Visu_Adv_Arr[2] := FALSE;
   S704_TL_DC_1ST_CLAMP1.Visu_Adv_Arr[3] := FALSE;
   S704_TL_DC_1ST_CLAMP1.Visu_Adv_Arr[4] := FALSE;
   S704_TL_DC_1ST_CLAMP1.Visu_Adv_Arr[5] := FALSE;
   S704_TL_DC_1ST_CLAMP1.Visu_Adv_Arr[6] := FALSE;
   S704_TL_DC_1ST_CLAMP1.Visu_Adv_Arr[7] := FALSE;
   S704_TL_DC_1ST_CLAMP1.Visu_Adv_Arr[8] := FALSE;
   S704_TL_DC_1ST_CLAMP1.Visu_Adv_Arr[9] := FALSE;
   S704_TL_DC_1ST_CLAMP1.Visu_Adv_Arr[10] := FALSE;
   S704_TL_DC_1ST_CLAMP1.Visu_Adv_Arr[11] := FALSE;
   S704_TL_DC_1ST_CLAMP1.Visu_Adv_Arr[12] := FALSE;
   S704_TL_DC_1ST_CLAMP1.Visu_Adv_Arr[13] := FALSE;
   S704_TL_DC_1ST_CLAMP1.Visu_Adv_Arr[14] := FALSE;
   S704_TL_DC_1ST_CLAMP1.Visu_Adv_Arr[15] := FALSE;
   S704_TL_DC_1ST_CLAMP1.Visu_Ret_Arr[0] := FALSE;
   S704_TL_DC_1ST_CLAMP1.Visu_Ret_Arr[1] := FALSE;
   S704_TL_DC_1ST_CLAMP1.Visu_Ret_Arr[2] := FALSE;
   S704_TL_DC_1ST_CLAMP1.Visu_Ret_Arr[3] := FALSE;
   S704_TL_DC_1ST_CLAMP1.Visu_Ret_Arr[4] := FALSE;
   S704_TL_DC_1ST_CLAMP1.Visu_Ret_Arr[5] := FALSE;
   S704_TL_DC_1ST_CLAMP1.Visu_Ret_Arr[6] := FALSE;
   S704_TL_DC_1ST_CLAMP1.Visu_Ret_Arr[7] := FALSE;
   S704_TL_DC_1ST_CLAMP1.Visu_Ret_Arr[8] := FALSE;
   S704_TL_DC_1ST_CLAMP1.Visu_Ret_Arr[9] := FALSE;
   S704_TL_DC_1ST_CLAMP1.Visu_Ret_Arr[10] := FALSE;
   S704_TL_DC_1ST_CLAMP1.Visu_Ret_Arr[11] := FALSE;
   S704_TL_DC_1ST_CLAMP1.Visu_Ret_Arr[12] := FALSE;
   S704_TL_DC_1ST_CLAMP1.Visu_Ret_Arr[13] := FALSE;
   S704_TL_DC_1ST_CLAMP1.Visu_Ret_Arr[14] := FALSE;
   S704_TL_DC_1ST_CLAMP1.Visu_Ret_Arr[15] := FALSE;
   S704_TL_DC_1ST_CLAMP1.BLK_Move_Ret := 0;
   S704_TL_DC_1ST_CLAMP1.Enable := FALSE;
   S704_TL_DC_1ST_CLAMP1.Adv_End := FALSE;
   S704_TL_DC_1ST_CLAMP1.Ret_End := FALSE;
   S704_TL_DC_1ST_CLAMP2.Enable_Aux := FALSE;
   S704_TL_DC_1ST_CLAMP2.Adv_Amount := 0;
   S704_TL_DC_1ST_CLAMP2.Ret_Amount := 0;
   S704_TL_DC_1ST_CLAMP2.LS_Adv1 := FALSE;
   S704_TL_DC_1ST_CLAMP2.LS_Ret1 := FALSE;
   S704_TL_DC_1ST_CLAMP2.LS_Adv2 := FALSE;
   S704_TL_DC_1ST_CLAMP2.LS_Ret2 := FALSE;
   S704_TL_DC_1ST_CLAMP2.LS_Adv3 := FALSE;
   S704_TL_DC_1ST_CLAMP2.LS_Ret3 := FALSE;
   S704_TL_DC_1ST_CLAMP2.LS_Adv4 := FALSE;
   S704_TL_DC_1ST_CLAMP2.LS_Ret4 := FALSE;
   S704_TL_DC_1ST_CLAMP2.LS_Adv5 := FALSE;
   S704_TL_DC_1ST_CLAMP2.LS_Ret5 := FALSE;
   S704_TL_DC_1ST_CLAMP2.LS_Adv6 := FALSE;
   S704_TL_DC_1ST_CLAMP2.LS_Ret6 := FALSE;
   S704_TL_DC_1ST_CLAMP2.LS_Adv7 := FALSE;
   S704_TL_DC_1ST_CLAMP2.LS_Ret7 := FALSE;
   S704_TL_DC_1ST_CLAMP2.LS_Adv8 := FALSE;
   S704_TL_DC_1ST_CLAMP2.LS_Ret8 := FALSE;
   S704_TL_DC_1ST_CLAMP2.SOL_Adv := FALSE;
   S704_TL_DC_1ST_CLAMP2.SOL_Ret := FALSE;
   S704_TL_DC_1ST_CLAMP2.M_Ready := FALSE;
   S704_TL_DC_1ST_CLAMP2.T_CHK1 := T#0MS;
   S704_TL_DC_1ST_CLAMP2.T_CHK2 := T#0MS;
   S704_TL_DC_1ST_CLAMP2.PB_Lamp_CHK := FALSE;
   S704_TL_DC_1ST_CLAMP2.PB_Error_Rst := FALSE;
   S704_TL_DC_1ST_CLAMP2.M_FLICK := FALSE;
   S704_TL_DC_1ST_CLAMP2.M_Adv_Err := FALSE;
   S704_TL_DC_1ST_CLAMP2.M_Ret_Err := FALSE;
   S704_TL_DC_1ST_CLAMP2.LP_Adv := FALSE;
   S704_TL_DC_1ST_CLAMP2.LP_Ret := FALSE;
   S704_TL_DC_1ST_CLAMP2.Visu_Adv := W#16#0;
   S704_TL_DC_1ST_CLAMP2.Visu_Ret := W#16#0;
   S704_TL_DC_1ST_CLAMP2.Error_T1.IN := FALSE;
   S704_TL_DC_1ST_CLAMP2.Error_T1.PT := T#0MS;
   S704_TL_DC_1ST_CLAMP2.Error_T1.Q := FALSE;
   S704_TL_DC_1ST_CLAMP2.Error_T1.ET := T#0MS;
   S704_TL_DC_1ST_CLAMP2.Error_T1.STATE := B#16#0;
   S704_TL_DC_1ST_CLAMP2.Error_T1.STIME := T#0MS;
   S704_TL_DC_1ST_CLAMP2.Error_T1.ATIME := T#0MS;
   S704_TL_DC_1ST_CLAMP2.Error_T2.IN := FALSE;
   S704_TL_DC_1ST_CLAMP2.Error_T2.PT := T#0MS;
   S704_TL_DC_1ST_CLAMP2.Error_T2.Q := FALSE;
   S704_TL_DC_1ST_CLAMP2.Error_T2.ET := T#0MS;
   S704_TL_DC_1ST_CLAMP2.Error_T2.STATE := B#16#0;
   S704_TL_DC_1ST_CLAMP2.Error_T2.STIME := T#0MS;
   S704_TL_DC_1ST_CLAMP2.Error_T2.ATIME := T#0MS;
   S704_TL_DC_1ST_CLAMP2.Adv_End_Aux := FALSE;
   S704_TL_DC_1ST_CLAMP2.Ret_End_Aux := FALSE;
   S704_TL_DC_1ST_CLAMP2.CHK_Aux1 := FALSE;
   S704_TL_DC_1ST_CLAMP2.CHK_Aux2 := FALSE;
   S704_TL_DC_1ST_CLAMP2.Error_T1_DN := FALSE;
   S704_TL_DC_1ST_CLAMP2.Error_T2_DN := FALSE;
   S704_TL_DC_1ST_CLAMP2.Adv_Memo := FALSE;
   S704_TL_DC_1ST_CLAMP2.Visu_Adv_Arr[0] := FALSE;
   S704_TL_DC_1ST_CLAMP2.Visu_Adv_Arr[1] := FALSE;
   S704_TL_DC_1ST_CLAMP2.Visu_Adv_Arr[2] := FALSE;
   S704_TL_DC_1ST_CLAMP2.Visu_Adv_Arr[3] := FALSE;
   S704_TL_DC_1ST_CLAMP2.Visu_Adv_Arr[4] := FALSE;
   S704_TL_DC_1ST_CLAMP2.Visu_Adv_Arr[5] := FALSE;
   S704_TL_DC_1ST_CLAMP2.Visu_Adv_Arr[6] := FALSE;
   S704_TL_DC_1ST_CLAMP2.Visu_Adv_Arr[7] := FALSE;
   S704_TL_DC_1ST_CLAMP2.Visu_Adv_Arr[8] := FALSE;
   S704_TL_DC_1ST_CLAMP2.Visu_Adv_Arr[9] := FALSE;
   S704_TL_DC_1ST_CLAMP2.Visu_Adv_Arr[10] := FALSE;
   S704_TL_DC_1ST_CLAMP2.Visu_Adv_Arr[11] := FALSE;
   S704_TL_DC_1ST_CLAMP2.Visu_Adv_Arr[12] := FALSE;
   S704_TL_DC_1ST_CLAMP2.Visu_Adv_Arr[13] := FALSE;
   S704_TL_DC_1ST_CLAMP2.Visu_Adv_Arr[14] := FALSE;
   S704_TL_DC_1ST_CLAMP2.Visu_Adv_Arr[15] := FALSE;
   S704_TL_DC_1ST_CLAMP2.Visu_Ret_Arr[0] := FALSE;
   S704_TL_DC_1ST_CLAMP2.Visu_Ret_Arr[1] := FALSE;
   S704_TL_DC_1ST_CLAMP2.Visu_Ret_Arr[2] := FALSE;
   S704_TL_DC_1ST_CLAMP2.Visu_Ret_Arr[3] := FALSE;
   S704_TL_DC_1ST_CLAMP2.Visu_Ret_Arr[4] := FALSE;
   S704_TL_DC_1ST_CLAMP2.Visu_Ret_Arr[5] := FALSE;
   S704_TL_DC_1ST_CLAMP2.Visu_Ret_Arr[6] := FALSE;
   S704_TL_DC_1ST_CLAMP2.Visu_Ret_Arr[7] := FALSE;
   S704_TL_DC_1ST_CLAMP2.Visu_Ret_Arr[8] := FALSE;
   S704_TL_DC_1ST_CLAMP2.Visu_Ret_Arr[9] := FALSE;
   S704_TL_DC_1ST_CLAMP2.Visu_Ret_Arr[10] := FALSE;
   S704_TL_DC_1ST_CLAMP2.Visu_Ret_Arr[11] := FALSE;
   S704_TL_DC_1ST_CLAMP2.Visu_Ret_Arr[12] := FALSE;
   S704_TL_DC_1ST_CLAMP2.Visu_Ret_Arr[13] := FALSE;
   S704_TL_DC_1ST_CLAMP2.Visu_Ret_Arr[14] := FALSE;
   S704_TL_DC_1ST_CLAMP2.Visu_Ret_Arr[15] := FALSE;
   S704_TL_DC_1ST_CLAMP2.BLK_Move_Ret := 0;
   S704_TL_DC_1ST_CLAMP2.Enable := FALSE;
   S704_TL_DC_1ST_CLAMP2.Adv_End := FALSE;
   S704_TL_DC_1ST_CLAMP2.Ret_End := FALSE;
   S704_TL_DC_1ST_CLAMP3.Enable_Aux := FALSE;
   S704_TL_DC_1ST_CLAMP3.Adv_Amount := 0;
   S704_TL_DC_1ST_CLAMP3.Ret_Amount := 0;
   S704_TL_DC_1ST_CLAMP3.LS_Adv1 := FALSE;
   S704_TL_DC_1ST_CLAMP3.LS_Ret1 := FALSE;
   S704_TL_DC_1ST_CLAMP3.LS_Adv2 := FALSE;
   S704_TL_DC_1ST_CLAMP3.LS_Ret2 := FALSE;
   S704_TL_DC_1ST_CLAMP3.LS_Adv3 := FALSE;
   S704_TL_DC_1ST_CLAMP3.LS_Ret3 := FALSE;
   S704_TL_DC_1ST_CLAMP3.LS_Adv4 := FALSE;
   S704_TL_DC_1ST_CLAMP3.LS_Ret4 := FALSE;
   S704_TL_DC_1ST_CLAMP3.LS_Adv5 := FALSE;
   S704_TL_DC_1ST_CLAMP3.LS_Ret5 := FALSE;
   S704_TL_DC_1ST_CLAMP3.LS_Adv6 := FALSE;
   S704_TL_DC_1ST_CLAMP3.LS_Ret6 := FALSE;
   S704_TL_DC_1ST_CLAMP3.LS_Adv7 := FALSE;
   S704_TL_DC_1ST_CLAMP3.LS_Ret7 := FALSE;
   S704_TL_DC_1ST_CLAMP3.LS_Adv8 := FALSE;
   S704_TL_DC_1ST_CLAMP3.LS_Ret8 := FALSE;
   S704_TL_DC_1ST_CLAMP3.SOL_Adv := FALSE;
   S704_TL_DC_1ST_CLAMP3.SOL_Ret := FALSE;
   S704_TL_DC_1ST_CLAMP3.M_Ready := FALSE;
   S704_TL_DC_1ST_CLAMP3.T_CHK1 := T#0MS;
   S704_TL_DC_1ST_CLAMP3.T_CHK2 := T#0MS;
   S704_TL_DC_1ST_CLAMP3.PB_Lamp_CHK := FALSE;
   S704_TL_DC_1ST_CLAMP3.PB_Error_Rst := FALSE;
   S704_TL_DC_1ST_CLAMP3.M_FLICK := FALSE;
   S704_TL_DC_1ST_CLAMP3.M_Adv_Err := FALSE;
   S704_TL_DC_1ST_CLAMP3.M_Ret_Err := FALSE;
   S704_TL_DC_1ST_CLAMP3.LP_Adv := FALSE;
   S704_TL_DC_1ST_CLAMP3.LP_Ret := FALSE;
   S704_TL_DC_1ST_CLAMP3.Visu_Adv := W#16#0;
   S704_TL_DC_1ST_CLAMP3.Visu_Ret := W#16#0;
   S704_TL_DC_1ST_CLAMP3.Error_T1.IN := FALSE;
   S704_TL_DC_1ST_CLAMP3.Error_T1.PT := T#0MS;
   S704_TL_DC_1ST_CLAMP3.Error_T1.Q := FALSE;
   S704_TL_DC_1ST_CLAMP3.Error_T1.ET := T#0MS;
   S704_TL_DC_1ST_CLAMP3.Error_T1.STATE := B#16#0;
   S704_TL_DC_1ST_CLAMP3.Error_T1.STIME := T#0MS;
   S704_TL_DC_1ST_CLAMP3.Error_T1.ATIME := T#0MS;
   S704_TL_DC_1ST_CLAMP3.Error_T2.IN := FALSE;
   S704_TL_DC_1ST_CLAMP3.Error_T2.PT := T#0MS;
   S704_TL_DC_1ST_CLAMP3.Error_T2.Q := FALSE;
   S704_TL_DC_1ST_CLAMP3.Error_T2.ET := T#0MS;
   S704_TL_DC_1ST_CLAMP3.Error_T2.STATE := B#16#0;
   S704_TL_DC_1ST_CLAMP3.Error_T2.STIME := T#0MS;
   S704_TL_DC_1ST_CLAMP3.Error_T2.ATIME := T#0MS;
   S704_TL_DC_1ST_CLAMP3.Adv_End_Aux := FALSE;
   S704_TL_DC_1ST_CLAMP3.Ret_End_Aux := FALSE;
   S704_TL_DC_1ST_CLAMP3.CHK_Aux1 := FALSE;
   S704_TL_DC_1ST_CLAMP3.CHK_Aux2 := FALSE;
   S704_TL_DC_1ST_CLAMP3.Error_T1_DN := FALSE;
   S704_TL_DC_1ST_CLAMP3.Error_T2_DN := FALSE;
   S704_TL_DC_1ST_CLAMP3.Adv_Memo := FALSE;
   S704_TL_DC_1ST_CLAMP3.Visu_Adv_Arr[0] := FALSE;
   S704_TL_DC_1ST_CLAMP3.Visu_Adv_Arr[1] := FALSE;
   S704_TL_DC_1ST_CLAMP3.Visu_Adv_Arr[2] := FALSE;
   S704_TL_DC_1ST_CLAMP3.Visu_Adv_Arr[3] := FALSE;
   S704_TL_DC_1ST_CLAMP3.Visu_Adv_Arr[4] := FALSE;
   S704_TL_DC_1ST_CLAMP3.Visu_Adv_Arr[5] := FALSE;
   S704_TL_DC_1ST_CLAMP3.Visu_Adv_Arr[6] := FALSE;
   S704_TL_DC_1ST_CLAMP3.Visu_Adv_Arr[7] := FALSE;
   S704_TL_DC_1ST_CLAMP3.Visu_Adv_Arr[8] := FALSE;
   S704_TL_DC_1ST_CLAMP3.Visu_Adv_Arr[9] := FALSE;
   S704_TL_DC_1ST_CLAMP3.Visu_Adv_Arr[10] := FALSE;
   S704_TL_DC_1ST_CLAMP3.Visu_Adv_Arr[11] := FALSE;
   S704_TL_DC_1ST_CLAMP3.Visu_Adv_Arr[12] := FALSE;
   S704_TL_DC_1ST_CLAMP3.Visu_Adv_Arr[13] := FALSE;
   S704_TL_DC_1ST_CLAMP3.Visu_Adv_Arr[14] := FALSE;
   S704_TL_DC_1ST_CLAMP3.Visu_Adv_Arr[15] := FALSE;
   S704_TL_DC_1ST_CLAMP3.Visu_Ret_Arr[0] := FALSE;
   S704_TL_DC_1ST_CLAMP3.Visu_Ret_Arr[1] := FALSE;
   S704_TL_DC_1ST_CLAMP3.Visu_Ret_Arr[2] := FALSE;
   S704_TL_DC_1ST_CLAMP3.Visu_Ret_Arr[3] := FALSE;
   S704_TL_DC_1ST_CLAMP3.Visu_Ret_Arr[4] := FALSE;
   S704_TL_DC_1ST_CLAMP3.Visu_Ret_Arr[5] := FALSE;
   S704_TL_DC_1ST_CLAMP3.Visu_Ret_Arr[6] := FALSE;
   S704_TL_DC_1ST_CLAMP3.Visu_Ret_Arr[7] := FALSE;
   S704_TL_DC_1ST_CLAMP3.Visu_Ret_Arr[8] := FALSE;
   S704_TL_DC_1ST_CLAMP3.Visu_Ret_Arr[9] := FALSE;
   S704_TL_DC_1ST_CLAMP3.Visu_Ret_Arr[10] := FALSE;
   S704_TL_DC_1ST_CLAMP3.Visu_Ret_Arr[11] := FALSE;
   S704_TL_DC_1ST_CLAMP3.Visu_Ret_Arr[12] := FALSE;
   S704_TL_DC_1ST_CLAMP3.Visu_Ret_Arr[13] := FALSE;
   S704_TL_DC_1ST_CLAMP3.Visu_Ret_Arr[14] := FALSE;
   S704_TL_DC_1ST_CLAMP3.Visu_Ret_Arr[15] := FALSE;
   S704_TL_DC_1ST_CLAMP3.BLK_Move_Ret := 0;
   S704_TL_DC_1ST_CLAMP3.Enable := FALSE;
   S704_TL_DC_1ST_CLAMP3.Adv_End := FALSE;
   S704_TL_DC_1ST_CLAMP3.Ret_End := FALSE;
   S704_TL_DC_2ND_CLAMP1.Enable_Aux := FALSE;
   S704_TL_DC_2ND_CLAMP1.Adv_Amount := 0;
   S704_TL_DC_2ND_CLAMP1.Ret_Amount := 0;
   S704_TL_DC_2ND_CLAMP1.LS_Adv1 := FALSE;
   S704_TL_DC_2ND_CLAMP1.LS_Ret1 := FALSE;
   S704_TL_DC_2ND_CLAMP1.LS_Adv2 := FALSE;
   S704_TL_DC_2ND_CLAMP1.LS_Ret2 := FALSE;
   S704_TL_DC_2ND_CLAMP1.LS_Adv3 := FALSE;
   S704_TL_DC_2ND_CLAMP1.LS_Ret3 := FALSE;
   S704_TL_DC_2ND_CLAMP1.LS_Adv4 := FALSE;
   S704_TL_DC_2ND_CLAMP1.LS_Ret4 := FALSE;
   S704_TL_DC_2ND_CLAMP1.LS_Adv5 := FALSE;
   S704_TL_DC_2ND_CLAMP1.LS_Ret5 := FALSE;
   S704_TL_DC_2ND_CLAMP1.LS_Adv6 := FALSE;
   S704_TL_DC_2ND_CLAMP1.LS_Ret6 := FALSE;
   S704_TL_DC_2ND_CLAMP1.LS_Adv7 := FALSE;
   S704_TL_DC_2ND_CLAMP1.LS_Ret7 := FALSE;
   S704_TL_DC_2ND_CLAMP1.LS_Adv8 := FALSE;
   S704_TL_DC_2ND_CLAMP1.LS_Ret8 := FALSE;
   S704_TL_DC_2ND_CLAMP1.SOL_Adv := FALSE;
   S704_TL_DC_2ND_CLAMP1.SOL_Ret := FALSE;
   S704_TL_DC_2ND_CLAMP1.M_Ready := FALSE;
   S704_TL_DC_2ND_CLAMP1.T_CHK1 := T#0MS;
   S704_TL_DC_2ND_CLAMP1.T_CHK2 := T#0MS;
   S704_TL_DC_2ND_CLAMP1.PB_Lamp_CHK := FALSE;
   S704_TL_DC_2ND_CLAMP1.PB_Error_Rst := FALSE;
   S704_TL_DC_2ND_CLAMP1.M_FLICK := FALSE;
   S704_TL_DC_2ND_CLAMP1.M_Adv_Err := FALSE;
   S704_TL_DC_2ND_CLAMP1.M_Ret_Err := FALSE;
   S704_TL_DC_2ND_CLAMP1.LP_Adv := FALSE;
   S704_TL_DC_2ND_CLAMP1.LP_Ret := FALSE;
   S704_TL_DC_2ND_CLAMP1.Visu_Adv := W#16#0;
   S704_TL_DC_2ND_CLAMP1.Visu_Ret := W#16#0;
   S704_TL_DC_2ND_CLAMP1.Error_T1.IN := FALSE;
   S704_TL_DC_2ND_CLAMP1.Error_T1.PT := T#0MS;
   S704_TL_DC_2ND_CLAMP1.Error_T1.Q := FALSE;
   S704_TL_DC_2ND_CLAMP1.Error_T1.ET := T#0MS;
   S704_TL_DC_2ND_CLAMP1.Error_T1.STATE := B#16#0;
   S704_TL_DC_2ND_CLAMP1.Error_T1.STIME := T#0MS;
   S704_TL_DC_2ND_CLAMP1.Error_T1.ATIME := T#0MS;
   S704_TL_DC_2ND_CLAMP1.Error_T2.IN := FALSE;
   S704_TL_DC_2ND_CLAMP1.Error_T2.PT := T#0MS;
   S704_TL_DC_2ND_CLAMP1.Error_T2.Q := FALSE;
   S704_TL_DC_2ND_CLAMP1.Error_T2.ET := T#0MS;
   S704_TL_DC_2ND_CLAMP1.Error_T2.STATE := B#16#0;
   S704_TL_DC_2ND_CLAMP1.Error_T2.STIME := T#0MS;
   S704_TL_DC_2ND_CLAMP1.Error_T2.ATIME := T#0MS;
   S704_TL_DC_2ND_CLAMP1.Adv_End_Aux := FALSE;
   S704_TL_DC_2ND_CLAMP1.Ret_End_Aux := FALSE;
   S704_TL_DC_2ND_CLAMP1.CHK_Aux1 := FALSE;
   S704_TL_DC_2ND_CLAMP1.CHK_Aux2 := FALSE;
   S704_TL_DC_2ND_CLAMP1.Error_T1_DN := FALSE;
   S704_TL_DC_2ND_CLAMP1.Error_T2_DN := FALSE;
   S704_TL_DC_2ND_CLAMP1.Adv_Memo := FALSE;
   S704_TL_DC_2ND_CLAMP1.Visu_Adv_Arr[0] := FALSE;
   S704_TL_DC_2ND_CLAMP1.Visu_Adv_Arr[1] := FALSE;
   S704_TL_DC_2ND_CLAMP1.Visu_Adv_Arr[2] := FALSE;
   S704_TL_DC_2ND_CLAMP1.Visu_Adv_Arr[3] := FALSE;
   S704_TL_DC_2ND_CLAMP1.Visu_Adv_Arr[4] := FALSE;
   S704_TL_DC_2ND_CLAMP1.Visu_Adv_Arr[5] := FALSE;
   S704_TL_DC_2ND_CLAMP1.Visu_Adv_Arr[6] := FALSE;
   S704_TL_DC_2ND_CLAMP1.Visu_Adv_Arr[7] := FALSE;
   S704_TL_DC_2ND_CLAMP1.Visu_Adv_Arr[8] := FALSE;
   S704_TL_DC_2ND_CLAMP1.Visu_Adv_Arr[9] := FALSE;
   S704_TL_DC_2ND_CLAMP1.Visu_Adv_Arr[10] := FALSE;
   S704_TL_DC_2ND_CLAMP1.Visu_Adv_Arr[11] := FALSE;
   S704_TL_DC_2ND_CLAMP1.Visu_Adv_Arr[12] := FALSE;
   S704_TL_DC_2ND_CLAMP1.Visu_Adv_Arr[13] := FALSE;
   S704_TL_DC_2ND_CLAMP1.Visu_Adv_Arr[14] := FALSE;
   S704_TL_DC_2ND_CLAMP1.Visu_Adv_Arr[15] := FALSE;
   S704_TL_DC_2ND_CLAMP1.Visu_Ret_Arr[0] := FALSE;
   S704_TL_DC_2ND_CLAMP1.Visu_Ret_Arr[1] := FALSE;
   S704_TL_DC_2ND_CLAMP1.Visu_Ret_Arr[2] := FALSE;
   S704_TL_DC_2ND_CLAMP1.Visu_Ret_Arr[3] := FALSE;
   S704_TL_DC_2ND_CLAMP1.Visu_Ret_Arr[4] := FALSE;
   S704_TL_DC_2ND_CLAMP1.Visu_Ret_Arr[5] := FALSE;
   S704_TL_DC_2ND_CLAMP1.Visu_Ret_Arr[6] := FALSE;
   S704_TL_DC_2ND_CLAMP1.Visu_Ret_Arr[7] := FALSE;
   S704_TL_DC_2ND_CLAMP1.Visu_Ret_Arr[8] := FALSE;
   S704_TL_DC_2ND_CLAMP1.Visu_Ret_Arr[9] := FALSE;
   S704_TL_DC_2ND_CLAMP1.Visu_Ret_Arr[10] := FALSE;
   S704_TL_DC_2ND_CLAMP1.Visu_Ret_Arr[11] := FALSE;
   S704_TL_DC_2ND_CLAMP1.Visu_Ret_Arr[12] := FALSE;
   S704_TL_DC_2ND_CLAMP1.Visu_Ret_Arr[13] := FALSE;
   S704_TL_DC_2ND_CLAMP1.Visu_Ret_Arr[14] := FALSE;
   S704_TL_DC_2ND_CLAMP1.Visu_Ret_Arr[15] := FALSE;
   S704_TL_DC_2ND_CLAMP1.BLK_Move_Ret := 0;
   S704_TL_DC_2ND_CLAMP1.Enable := FALSE;
   S704_TL_DC_2ND_CLAMP1.Adv_End := FALSE;
   S704_TL_DC_2ND_CLAMP1.Ret_End := FALSE;
   S704_TL_DC_2ND_CLAMP2.Enable_Aux := FALSE;
   S704_TL_DC_2ND_CLAMP2.Adv_Amount := 0;
   S704_TL_DC_2ND_CLAMP2.Ret_Amount := 0;
   S704_TL_DC_2ND_CLAMP2.LS_Adv1 := FALSE;
   S704_TL_DC_2ND_CLAMP2.LS_Ret1 := FALSE;
   S704_TL_DC_2ND_CLAMP2.LS_Adv2 := FALSE;
   S704_TL_DC_2ND_CLAMP2.LS_Ret2 := FALSE;
   S704_TL_DC_2ND_CLAMP2.LS_Adv3 := FALSE;
   S704_TL_DC_2ND_CLAMP2.LS_Ret3 := FALSE;
   S704_TL_DC_2ND_CLAMP2.LS_Adv4 := FALSE;
   S704_TL_DC_2ND_CLAMP2.LS_Ret4 := FALSE;
   S704_TL_DC_2ND_CLAMP2.LS_Adv5 := FALSE;
   S704_TL_DC_2ND_CLAMP2.LS_Ret5 := FALSE;
   S704_TL_DC_2ND_CLAMP2.LS_Adv6 := FALSE;
   S704_TL_DC_2ND_CLAMP2.LS_Ret6 := FALSE;
   S704_TL_DC_2ND_CLAMP2.LS_Adv7 := FALSE;
   S704_TL_DC_2ND_CLAMP2.LS_Ret7 := FALSE;
   S704_TL_DC_2ND_CLAMP2.LS_Adv8 := FALSE;
   S704_TL_DC_2ND_CLAMP2.LS_Ret8 := FALSE;
   S704_TL_DC_2ND_CLAMP2.SOL_Adv := FALSE;
   S704_TL_DC_2ND_CLAMP2.SOL_Ret := FALSE;
   S704_TL_DC_2ND_CLAMP2.M_Ready := FALSE;
   S704_TL_DC_2ND_CLAMP2.T_CHK1 := T#0MS;
   S704_TL_DC_2ND_CLAMP2.T_CHK2 := T#0MS;
   S704_TL_DC_2ND_CLAMP2.PB_Lamp_CHK := FALSE;
   S704_TL_DC_2ND_CLAMP2.PB_Error_Rst := FALSE;
   S704_TL_DC_2ND_CLAMP2.M_FLICK := FALSE;
   S704_TL_DC_2ND_CLAMP2.M_Adv_Err := FALSE;
   S704_TL_DC_2ND_CLAMP2.M_Ret_Err := FALSE;
   S704_TL_DC_2ND_CLAMP2.LP_Adv := FALSE;
   S704_TL_DC_2ND_CLAMP2.LP_Ret := FALSE;
   S704_TL_DC_2ND_CLAMP2.Visu_Adv := W#16#0;
   S704_TL_DC_2ND_CLAMP2.Visu_Ret := W#16#0;
   S704_TL_DC_2ND_CLAMP2.Error_T1.IN := FALSE;
   S704_TL_DC_2ND_CLAMP2.Error_T1.PT := T#0MS;
   S704_TL_DC_2ND_CLAMP2.Error_T1.Q := FALSE;
   S704_TL_DC_2ND_CLAMP2.Error_T1.ET := T#0MS;
   S704_TL_DC_2ND_CLAMP2.Error_T1.STATE := B#16#0;
   S704_TL_DC_2ND_CLAMP2.Error_T1.STIME := T#0MS;
   S704_TL_DC_2ND_CLAMP2.Error_T1.ATIME := T#0MS;
   S704_TL_DC_2ND_CLAMP2.Error_T2.IN := FALSE;
   S704_TL_DC_2ND_CLAMP2.Error_T2.PT := T#0MS;
   S704_TL_DC_2ND_CLAMP2.Error_T2.Q := FALSE;
   S704_TL_DC_2ND_CLAMP2.Error_T2.ET := T#0MS;
   S704_TL_DC_2ND_CLAMP2.Error_T2.STATE := B#16#0;
   S704_TL_DC_2ND_CLAMP2.Error_T2.STIME := T#0MS;
   S704_TL_DC_2ND_CLAMP2.Error_T2.ATIME := T#0MS;
   S704_TL_DC_2ND_CLAMP2.Adv_End_Aux := FALSE;
   S704_TL_DC_2ND_CLAMP2.Ret_End_Aux := FALSE;
   S704_TL_DC_2ND_CLAMP2.CHK_Aux1 := FALSE;
   S704_TL_DC_2ND_CLAMP2.CHK_Aux2 := FALSE;
   S704_TL_DC_2ND_CLAMP2.Error_T1_DN := FALSE;
   S704_TL_DC_2ND_CLAMP2.Error_T2_DN := FALSE;
   S704_TL_DC_2ND_CLAMP2.Adv_Memo := FALSE;
   S704_TL_DC_2ND_CLAMP2.Visu_Adv_Arr[0] := FALSE;
   S704_TL_DC_2ND_CLAMP2.Visu_Adv_Arr[1] := FALSE;
   S704_TL_DC_2ND_CLAMP2.Visu_Adv_Arr[2] := FALSE;
   S704_TL_DC_2ND_CLAMP2.Visu_Adv_Arr[3] := FALSE;
   S704_TL_DC_2ND_CLAMP2.Visu_Adv_Arr[4] := FALSE;
   S704_TL_DC_2ND_CLAMP2.Visu_Adv_Arr[5] := FALSE;
   S704_TL_DC_2ND_CLAMP2.Visu_Adv_Arr[6] := FALSE;
   S704_TL_DC_2ND_CLAMP2.Visu_Adv_Arr[7] := FALSE;
   S704_TL_DC_2ND_CLAMP2.Visu_Adv_Arr[8] := FALSE;
   S704_TL_DC_2ND_CLAMP2.Visu_Adv_Arr[9] := FALSE;
   S704_TL_DC_2ND_CLAMP2.Visu_Adv_Arr[10] := FALSE;
   S704_TL_DC_2ND_CLAMP2.Visu_Adv_Arr[11] := FALSE;
   S704_TL_DC_2ND_CLAMP2.Visu_Adv_Arr[12] := FALSE;
   S704_TL_DC_2ND_CLAMP2.Visu_Adv_Arr[13] := FALSE;
   S704_TL_DC_2ND_CLAMP2.Visu_Adv_Arr[14] := FALSE;
   S704_TL_DC_2ND_CLAMP2.Visu_Adv_Arr[15] := FALSE;
   S704_TL_DC_2ND_CLAMP2.Visu_Ret_Arr[0] := FALSE;
   S704_TL_DC_2ND_CLAMP2.Visu_Ret_Arr[1] := FALSE;
   S704_TL_DC_2ND_CLAMP2.Visu_Ret_Arr[2] := FALSE;
   S704_TL_DC_2ND_CLAMP2.Visu_Ret_Arr[3] := FALSE;
   S704_TL_DC_2ND_CLAMP2.Visu_Ret_Arr[4] := FALSE;
   S704_TL_DC_2ND_CLAMP2.Visu_Ret_Arr[5] := FALSE;
   S704_TL_DC_2ND_CLAMP2.Visu_Ret_Arr[6] := FALSE;
   S704_TL_DC_2ND_CLAMP2.Visu_Ret_Arr[7] := FALSE;
   S704_TL_DC_2ND_CLAMP2.Visu_Ret_Arr[8] := FALSE;
   S704_TL_DC_2ND_CLAMP2.Visu_Ret_Arr[9] := FALSE;
   S704_TL_DC_2ND_CLAMP2.Visu_Ret_Arr[10] := FALSE;
   S704_TL_DC_2ND_CLAMP2.Visu_Ret_Arr[11] := FALSE;
   S704_TL_DC_2ND_CLAMP2.Visu_Ret_Arr[12] := FALSE;
   S704_TL_DC_2ND_CLAMP2.Visu_Ret_Arr[13] := FALSE;
   S704_TL_DC_2ND_CLAMP2.Visu_Ret_Arr[14] := FALSE;
   S704_TL_DC_2ND_CLAMP2.Visu_Ret_Arr[15] := FALSE;
   S704_TL_DC_2ND_CLAMP2.BLK_Move_Ret := 0;
   S704_TL_DC_2ND_CLAMP2.Enable := FALSE;
   S704_TL_DC_2ND_CLAMP2.Adv_End := FALSE;
   S704_TL_DC_2ND_CLAMP2.Ret_End := FALSE;
   S704_TL_DC_U261.Enable_Aux := FALSE;
   S704_TL_DC_U261.Adv_Amount := 0;
   S704_TL_DC_U261.Ret_Amount := 0;
   S704_TL_DC_U261.LS_Adv1 := FALSE;
   S704_TL_DC_U261.LS_Ret1 := FALSE;
   S704_TL_DC_U261.LS_Adv2 := FALSE;
   S704_TL_DC_U261.LS_Ret2 := FALSE;
   S704_TL_DC_U261.LS_Adv3 := FALSE;
   S704_TL_DC_U261.LS_Ret3 := FALSE;
   S704_TL_DC_U261.LS_Adv4 := FALSE;
   S704_TL_DC_U261.LS_Ret4 := FALSE;
   S704_TL_DC_U261.LS_Adv5 := FALSE;
   S704_TL_DC_U261.LS_Ret5 := FALSE;
   S704_TL_DC_U261.LS_Adv6 := FALSE;
   S704_TL_DC_U261.LS_Ret6 := FALSE;
   S704_TL_DC_U261.LS_Adv7 := FALSE;
   S704_TL_DC_U261.LS_Ret7 := FALSE;
   S704_TL_DC_U261.LS_Adv8 := FALSE;
   S704_TL_DC_U261.LS_Ret8 := FALSE;
   S704_TL_DC_U261.SOL_Adv := FALSE;
   S704_TL_DC_U261.SOL_Ret := FALSE;
   S704_TL_DC_U261.M_Ready := FALSE;
   S704_TL_DC_U261.T_CHK1 := T#0MS;
   S704_TL_DC_U261.T_CHK2 := T#0MS;
   S704_TL_DC_U261.PB_Lamp_CHK := FALSE;
   S704_TL_DC_U261.PB_Error_Rst := FALSE;
   S704_TL_DC_U261.M_FLICK := FALSE;
   S704_TL_DC_U261.M_Adv_Err := FALSE;
   S704_TL_DC_U261.M_Ret_Err := FALSE;
   S704_TL_DC_U261.LP_Adv := FALSE;
   S704_TL_DC_U261.LP_Ret := FALSE;
   S704_TL_DC_U261.Visu_Adv := W#16#0;
   S704_TL_DC_U261.Visu_Ret := W#16#0;
   S704_TL_DC_U261.Error_T1.IN := FALSE;
   S704_TL_DC_U261.Error_T1.PT := T#0MS;
   S704_TL_DC_U261.Error_T1.Q := FALSE;
   S704_TL_DC_U261.Error_T1.ET := T#0MS;
   S704_TL_DC_U261.Error_T1.STATE := B#16#0;
   S704_TL_DC_U261.Error_T1.STIME := T#0MS;
   S704_TL_DC_U261.Error_T1.ATIME := T#0MS;
   S704_TL_DC_U261.Error_T2.IN := FALSE;
   S704_TL_DC_U261.Error_T2.PT := T#0MS;
   S704_TL_DC_U261.Error_T2.Q := FALSE;
   S704_TL_DC_U261.Error_T2.ET := T#0MS;
   S704_TL_DC_U261.Error_T2.STATE := B#16#0;
   S704_TL_DC_U261.Error_T2.STIME := T#0MS;
   S704_TL_DC_U261.Error_T2.ATIME := T#0MS;
   S704_TL_DC_U261.Adv_End_Aux := FALSE;
   S704_TL_DC_U261.Ret_End_Aux := FALSE;
   S704_TL_DC_U261.CHK_Aux1 := FALSE;
   S704_TL_DC_U261.CHK_Aux2 := FALSE;
   S704_TL_DC_U261.Error_T1_DN := FALSE;
   S704_TL_DC_U261.Error_T2_DN := FALSE;
   S704_TL_DC_U261.Adv_Memo := FALSE;
   S704_TL_DC_U261.Visu_Adv_Arr[0] := FALSE;
   S704_TL_DC_U261.Visu_Adv_Arr[1] := FALSE;
   S704_TL_DC_U261.Visu_Adv_Arr[2] := FALSE;
   S704_TL_DC_U261.Visu_Adv_Arr[3] := FALSE;
   S704_TL_DC_U261.Visu_Adv_Arr[4] := FALSE;
   S704_TL_DC_U261.Visu_Adv_Arr[5] := FALSE;
   S704_TL_DC_U261.Visu_Adv_Arr[6] := FALSE;
   S704_TL_DC_U261.Visu_Adv_Arr[7] := FALSE;
   S704_TL_DC_U261.Visu_Adv_Arr[8] := FALSE;
   S704_TL_DC_U261.Visu_Adv_Arr[9] := FALSE;
   S704_TL_DC_U261.Visu_Adv_Arr[10] := FALSE;
   S704_TL_DC_U261.Visu_Adv_Arr[11] := FALSE;
   S704_TL_DC_U261.Visu_Adv_Arr[12] := FALSE;
   S704_TL_DC_U261.Visu_Adv_Arr[13] := FALSE;
   S704_TL_DC_U261.Visu_Adv_Arr[14] := FALSE;
   S704_TL_DC_U261.Visu_Adv_Arr[15] := FALSE;
   S704_TL_DC_U261.Visu_Ret_Arr[0] := FALSE;
   S704_TL_DC_U261.Visu_Ret_Arr[1] := FALSE;
   S704_TL_DC_U261.Visu_Ret_Arr[2] := FALSE;
   S704_TL_DC_U261.Visu_Ret_Arr[3] := FALSE;
   S704_TL_DC_U261.Visu_Ret_Arr[4] := FALSE;
   S704_TL_DC_U261.Visu_Ret_Arr[5] := FALSE;
   S704_TL_DC_U261.Visu_Ret_Arr[6] := FALSE;
   S704_TL_DC_U261.Visu_Ret_Arr[7] := FALSE;
   S704_TL_DC_U261.Visu_Ret_Arr[8] := FALSE;
   S704_TL_DC_U261.Visu_Ret_Arr[9] := FALSE;
   S704_TL_DC_U261.Visu_Ret_Arr[10] := FALSE;
   S704_TL_DC_U261.Visu_Ret_Arr[11] := FALSE;
   S704_TL_DC_U261.Visu_Ret_Arr[12] := FALSE;
   S704_TL_DC_U261.Visu_Ret_Arr[13] := FALSE;
   S704_TL_DC_U261.Visu_Ret_Arr[14] := FALSE;
   S704_TL_DC_U261.Visu_Ret_Arr[15] := FALSE;
   S704_TL_DC_U261.BLK_Move_Ret := 0;
   S704_TL_DC_U261.Enable := FALSE;
   S704_TL_DC_U261.Adv_End := FALSE;
   S704_TL_DC_U261.Ret_End := FALSE;
   S704_TL_DC_U261_CLAMP.Enable_Aux := FALSE;
   S704_TL_DC_U261_CLAMP.Adv_Amount := 0;
   S704_TL_DC_U261_CLAMP.Ret_Amount := 0;
   S704_TL_DC_U261_CLAMP.LS_Adv1 := FALSE;
   S704_TL_DC_U261_CLAMP.LS_Ret1 := FALSE;
   S704_TL_DC_U261_CLAMP.LS_Adv2 := FALSE;
   S704_TL_DC_U261_CLAMP.LS_Ret2 := FALSE;
   S704_TL_DC_U261_CLAMP.LS_Adv3 := FALSE;
   S704_TL_DC_U261_CLAMP.LS_Ret3 := FALSE;
   S704_TL_DC_U261_CLAMP.LS_Adv4 := FALSE;
   S704_TL_DC_U261_CLAMP.LS_Ret4 := FALSE;
   S704_TL_DC_U261_CLAMP.LS_Adv5 := FALSE;
   S704_TL_DC_U261_CLAMP.LS_Ret5 := FALSE;
   S704_TL_DC_U261_CLAMP.LS_Adv6 := FALSE;
   S704_TL_DC_U261_CLAMP.LS_Ret6 := FALSE;
   S704_TL_DC_U261_CLAMP.LS_Adv7 := FALSE;
   S704_TL_DC_U261_CLAMP.LS_Ret7 := FALSE;
   S704_TL_DC_U261_CLAMP.LS_Adv8 := FALSE;
   S704_TL_DC_U261_CLAMP.LS_Ret8 := FALSE;
   S704_TL_DC_U261_CLAMP.SOL_Adv := FALSE;
   S704_TL_DC_U261_CLAMP.SOL_Ret := FALSE;
   S704_TL_DC_U261_CLAMP.M_Ready := FALSE;
   S704_TL_DC_U261_CLAMP.T_CHK1 := T#0MS;
   S704_TL_DC_U261_CLAMP.T_CHK2 := T#0MS;
   S704_TL_DC_U261_CLAMP.PB_Lamp_CHK := FALSE;
   S704_TL_DC_U261_CLAMP.PB_Error_Rst := FALSE;
   S704_TL_DC_U261_CLAMP.M_FLICK := FALSE;
   S704_TL_DC_U261_CLAMP.M_Adv_Err := FALSE;
   S704_TL_DC_U261_CLAMP.M_Ret_Err := FALSE;
   S704_TL_DC_U261_CLAMP.LP_Adv := FALSE;
   S704_TL_DC_U261_CLAMP.LP_Ret := FALSE;
   S704_TL_DC_U261_CLAMP.Visu_Adv := W#16#0;
   S704_TL_DC_U261_CLAMP.Visu_Ret := W#16#0;
   S704_TL_DC_U261_CLAMP.Error_T1.IN := FALSE;
   S704_TL_DC_U261_CLAMP.Error_T1.PT := T#0MS;
   S704_TL_DC_U261_CLAMP.Error_T1.Q := FALSE;
   S704_TL_DC_U261_CLAMP.Error_T1.ET := T#0MS;
   S704_TL_DC_U261_CLAMP.Error_T1.STATE := B#16#0;
   S704_TL_DC_U261_CLAMP.Error_T1.STIME := T#0MS;
   S704_TL_DC_U261_CLAMP.Error_T1.ATIME := T#0MS;
   S704_TL_DC_U261_CLAMP.Error_T2.IN := FALSE;
   S704_TL_DC_U261_CLAMP.Error_T2.PT := T#0MS;
   S704_TL_DC_U261_CLAMP.Error_T2.Q := FALSE;
   S704_TL_DC_U261_CLAMP.Error_T2.ET := T#0MS;
   S704_TL_DC_U261_CLAMP.Error_T2.STATE := B#16#0;
   S704_TL_DC_U261_CLAMP.Error_T2.STIME := T#0MS;
   S704_TL_DC_U261_CLAMP.Error_T2.ATIME := T#0MS;
   S704_TL_DC_U261_CLAMP.Adv_End_Aux := FALSE;
   S704_TL_DC_U261_CLAMP.Ret_End_Aux := FALSE;
   S704_TL_DC_U261_CLAMP.CHK_Aux1 := FALSE;
   S704_TL_DC_U261_CLAMP.CHK_Aux2 := FALSE;
   S704_TL_DC_U261_CLAMP.Error_T1_DN := FALSE;
   S704_TL_DC_U261_CLAMP.Error_T2_DN := FALSE;
   S704_TL_DC_U261_CLAMP.Adv_Memo := FALSE;
   S704_TL_DC_U261_CLAMP.Visu_Adv_Arr[0] := FALSE;
   S704_TL_DC_U261_CLAMP.Visu_Adv_Arr[1] := FALSE;
   S704_TL_DC_U261_CLAMP.Visu_Adv_Arr[2] := FALSE;
   S704_TL_DC_U261_CLAMP.Visu_Adv_Arr[3] := FALSE;
   S704_TL_DC_U261_CLAMP.Visu_Adv_Arr[4] := FALSE;
   S704_TL_DC_U261_CLAMP.Visu_Adv_Arr[5] := FALSE;
   S704_TL_DC_U261_CLAMP.Visu_Adv_Arr[6] := FALSE;
   S704_TL_DC_U261_CLAMP.Visu_Adv_Arr[7] := FALSE;
   S704_TL_DC_U261_CLAMP.Visu_Adv_Arr[8] := FALSE;
   S704_TL_DC_U261_CLAMP.Visu_Adv_Arr[9] := FALSE;
   S704_TL_DC_U261_CLAMP.Visu_Adv_Arr[10] := FALSE;
   S704_TL_DC_U261_CLAMP.Visu_Adv_Arr[11] := FALSE;
   S704_TL_DC_U261_CLAMP.Visu_Adv_Arr[12] := FALSE;
   S704_TL_DC_U261_CLAMP.Visu_Adv_Arr[13] := FALSE;
   S704_TL_DC_U261_CLAMP.Visu_Adv_Arr[14] := FALSE;
   S704_TL_DC_U261_CLAMP.Visu_Adv_Arr[15] := FALSE;
   S704_TL_DC_U261_CLAMP.Visu_Ret_Arr[0] := FALSE;
   S704_TL_DC_U261_CLAMP.Visu_Ret_Arr[1] := FALSE;
   S704_TL_DC_U261_CLAMP.Visu_Ret_Arr[2] := FALSE;
   S704_TL_DC_U261_CLAMP.Visu_Ret_Arr[3] := FALSE;
   S704_TL_DC_U261_CLAMP.Visu_Ret_Arr[4] := FALSE;
   S704_TL_DC_U261_CLAMP.Visu_Ret_Arr[5] := FALSE;
   S704_TL_DC_U261_CLAMP.Visu_Ret_Arr[6] := FALSE;
   S704_TL_DC_U261_CLAMP.Visu_Ret_Arr[7] := FALSE;
   S704_TL_DC_U261_CLAMP.Visu_Ret_Arr[8] := FALSE;
   S704_TL_DC_U261_CLAMP.Visu_Ret_Arr[9] := FALSE;
   S704_TL_DC_U261_CLAMP.Visu_Ret_Arr[10] := FALSE;
   S704_TL_DC_U261_CLAMP.Visu_Ret_Arr[11] := FALSE;
   S704_TL_DC_U261_CLAMP.Visu_Ret_Arr[12] := FALSE;
   S704_TL_DC_U261_CLAMP.Visu_Ret_Arr[13] := FALSE;
   S704_TL_DC_U261_CLAMP.Visu_Ret_Arr[14] := FALSE;
   S704_TL_DC_U261_CLAMP.Visu_Ret_Arr[15] := FALSE;
   S704_TL_DC_U261_CLAMP.BLK_Move_Ret := 0;
   S704_TL_DC_U261_CLAMP.Enable := FALSE;
   S704_TL_DC_U261_CLAMP.Adv_End := FALSE;
   S704_TL_DC_U261_CLAMP.Ret_End := FALSE;
   S704_TL_DC_U269.Enable_Aux := FALSE;
   S704_TL_DC_U269.Adv_Amount := 0;
   S704_TL_DC_U269.Ret_Amount := 0;
   S704_TL_DC_U269.LS_Adv1 := FALSE;
   S704_TL_DC_U269.LS_Ret1 := FALSE;
   S704_TL_DC_U269.LS_Adv2 := FALSE;
   S704_TL_DC_U269.LS_Ret2 := FALSE;
   S704_TL_DC_U269.LS_Adv3 := FALSE;
   S704_TL_DC_U269.LS_Ret3 := FALSE;
   S704_TL_DC_U269.LS_Adv4 := FALSE;
   S704_TL_DC_U269.LS_Ret4 := FALSE;
   S704_TL_DC_U269.LS_Adv5 := FALSE;
   S704_TL_DC_U269.LS_Ret5 := FALSE;
   S704_TL_DC_U269.LS_Adv6 := FALSE;
   S704_TL_DC_U269.LS_Ret6 := FALSE;
   S704_TL_DC_U269.LS_Adv7 := FALSE;
   S704_TL_DC_U269.LS_Ret7 := FALSE;
   S704_TL_DC_U269.LS_Adv8 := FALSE;
   S704_TL_DC_U269.LS_Ret8 := FALSE;
   S704_TL_DC_U269.SOL_Adv := FALSE;
   S704_TL_DC_U269.SOL_Ret := FALSE;
   S704_TL_DC_U269.M_Ready := FALSE;
   S704_TL_DC_U269.T_CHK1 := T#0MS;
   S704_TL_DC_U269.T_CHK2 := T#0MS;
   S704_TL_DC_U269.PB_Lamp_CHK := FALSE;
   S704_TL_DC_U269.PB_Error_Rst := FALSE;
   S704_TL_DC_U269.M_FLICK := FALSE;
   S704_TL_DC_U269.M_Adv_Err := FALSE;
   S704_TL_DC_U269.M_Ret_Err := FALSE;
   S704_TL_DC_U269.LP_Adv := FALSE;
   S704_TL_DC_U269.LP_Ret := FALSE;
   S704_TL_DC_U269.Visu_Adv := W#16#0;
   S704_TL_DC_U269.Visu_Ret := W#16#0;
   S704_TL_DC_U269.Error_T1.IN := FALSE;
   S704_TL_DC_U269.Error_T1.PT := T#0MS;
   S704_TL_DC_U269.Error_T1.Q := FALSE;
   S704_TL_DC_U269.Error_T1.ET := T#0MS;
   S704_TL_DC_U269.Error_T1.STATE := B#16#0;
   S704_TL_DC_U269.Error_T1.STIME := T#0MS;
   S704_TL_DC_U269.Error_T1.ATIME := T#0MS;
   S704_TL_DC_U269.Error_T2.IN := FALSE;
   S704_TL_DC_U269.Error_T2.PT := T#0MS;
   S704_TL_DC_U269.Error_T2.Q := FALSE;
   S704_TL_DC_U269.Error_T2.ET := T#0MS;
   S704_TL_DC_U269.Error_T2.STATE := B#16#0;
   S704_TL_DC_U269.Error_T2.STIME := T#0MS;
   S704_TL_DC_U269.Error_T2.ATIME := T#0MS;
   S704_TL_DC_U269.Adv_End_Aux := FALSE;
   S704_TL_DC_U269.Ret_End_Aux := FALSE;
   S704_TL_DC_U269.CHK_Aux1 := FALSE;
   S704_TL_DC_U269.CHK_Aux2 := FALSE;
   S704_TL_DC_U269.Error_T1_DN := FALSE;
   S704_TL_DC_U269.Error_T2_DN := FALSE;
   S704_TL_DC_U269.Adv_Memo := FALSE;
   S704_TL_DC_U269.Visu_Adv_Arr[0] := FALSE;
   S704_TL_DC_U269.Visu_Adv_Arr[1] := FALSE;
   S704_TL_DC_U269.Visu_Adv_Arr[2] := FALSE;
   S704_TL_DC_U269.Visu_Adv_Arr[3] := FALSE;
   S704_TL_DC_U269.Visu_Adv_Arr[4] := FALSE;
   S704_TL_DC_U269.Visu_Adv_Arr[5] := FALSE;
   S704_TL_DC_U269.Visu_Adv_Arr[6] := FALSE;
   S704_TL_DC_U269.Visu_Adv_Arr[7] := FALSE;
   S704_TL_DC_U269.Visu_Adv_Arr[8] := FALSE;
   S704_TL_DC_U269.Visu_Adv_Arr[9] := FALSE;
   S704_TL_DC_U269.Visu_Adv_Arr[10] := FALSE;
   S704_TL_DC_U269.Visu_Adv_Arr[11] := FALSE;
   S704_TL_DC_U269.Visu_Adv_Arr[12] := FALSE;
   S704_TL_DC_U269.Visu_Adv_Arr[13] := FALSE;
   S704_TL_DC_U269.Visu_Adv_Arr[14] := FALSE;
   S704_TL_DC_U269.Visu_Adv_Arr[15] := FALSE;
   S704_TL_DC_U269.Visu_Ret_Arr[0] := FALSE;
   S704_TL_DC_U269.Visu_Ret_Arr[1] := FALSE;
   S704_TL_DC_U269.Visu_Ret_Arr[2] := FALSE;
   S704_TL_DC_U269.Visu_Ret_Arr[3] := FALSE;
   S704_TL_DC_U269.Visu_Ret_Arr[4] := FALSE;
   S704_TL_DC_U269.Visu_Ret_Arr[5] := FALSE;
   S704_TL_DC_U269.Visu_Ret_Arr[6] := FALSE;
   S704_TL_DC_U269.Visu_Ret_Arr[7] := FALSE;
   S704_TL_DC_U269.Visu_Ret_Arr[8] := FALSE;
   S704_TL_DC_U269.Visu_Ret_Arr[9] := FALSE;
   S704_TL_DC_U269.Visu_Ret_Arr[10] := FALSE;
   S704_TL_DC_U269.Visu_Ret_Arr[11] := FALSE;
   S704_TL_DC_U269.Visu_Ret_Arr[12] := FALSE;
   S704_TL_DC_U269.Visu_Ret_Arr[13] := FALSE;
   S704_TL_DC_U269.Visu_Ret_Arr[14] := FALSE;
   S704_TL_DC_U269.Visu_Ret_Arr[15] := FALSE;
   S704_TL_DC_U269.BLK_Move_Ret := 0;
   S704_TL_DC_U269.Enable := FALSE;
   S704_TL_DC_U269.Adv_End := FALSE;
   S704_TL_DC_U269.Ret_End := FALSE;
   S704_TL_DC_U269_CLAMP.Enable_Aux := FALSE;
   S704_TL_DC_U269_CLAMP.Adv_Amount := 0;
   S704_TL_DC_U269_CLAMP.Ret_Amount := 0;
   S704_TL_DC_U269_CLAMP.LS_Adv1 := FALSE;
   S704_TL_DC_U269_CLAMP.LS_Ret1 := FALSE;
   S704_TL_DC_U269_CLAMP.LS_Adv2 := FALSE;
   S704_TL_DC_U269_CLAMP.LS_Ret2 := FALSE;
   S704_TL_DC_U269_CLAMP.LS_Adv3 := FALSE;
   S704_TL_DC_U269_CLAMP.LS_Ret3 := FALSE;
   S704_TL_DC_U269_CLAMP.LS_Adv4 := FALSE;
   S704_TL_DC_U269_CLAMP.LS_Ret4 := FALSE;
   S704_TL_DC_U269_CLAMP.LS_Adv5 := FALSE;
   S704_TL_DC_U269_CLAMP.LS_Ret5 := FALSE;
   S704_TL_DC_U269_CLAMP.LS_Adv6 := FALSE;
   S704_TL_DC_U269_CLAMP.LS_Ret6 := FALSE;
   S704_TL_DC_U269_CLAMP.LS_Adv7 := FALSE;
   S704_TL_DC_U269_CLAMP.LS_Ret7 := FALSE;
   S704_TL_DC_U269_CLAMP.LS_Adv8 := FALSE;
   S704_TL_DC_U269_CLAMP.LS_Ret8 := FALSE;
   S704_TL_DC_U269_CLAMP.SOL_Adv := FALSE;
   S704_TL_DC_U269_CLAMP.SOL_Ret := FALSE;
   S704_TL_DC_U269_CLAMP.M_Ready := FALSE;
   S704_TL_DC_U269_CLAMP.T_CHK1 := T#0MS;
   S704_TL_DC_U269_CLAMP.T_CHK2 := T#0MS;
   S704_TL_DC_U269_CLAMP.PB_Lamp_CHK := FALSE;
   S704_TL_DC_U269_CLAMP.PB_Error_Rst := FALSE;
   S704_TL_DC_U269_CLAMP.M_FLICK := FALSE;
   S704_TL_DC_U269_CLAMP.M_Adv_Err := FALSE;
   S704_TL_DC_U269_CLAMP.M_Ret_Err := FALSE;
   S704_TL_DC_U269_CLAMP.LP_Adv := FALSE;
   S704_TL_DC_U269_CLAMP.LP_Ret := FALSE;
   S704_TL_DC_U269_CLAMP.Visu_Adv := W#16#0;
   S704_TL_DC_U269_CLAMP.Visu_Ret := W#16#0;
   S704_TL_DC_U269_CLAMP.Error_T1.IN := FALSE;
   S704_TL_DC_U269_CLAMP.Error_T1.PT := T#0MS;
   S704_TL_DC_U269_CLAMP.Error_T1.Q := FALSE;
   S704_TL_DC_U269_CLAMP.Error_T1.ET := T#0MS;
   S704_TL_DC_U269_CLAMP.Error_T1.STATE := B#16#0;
   S704_TL_DC_U269_CLAMP.Error_T1.STIME := T#0MS;
   S704_TL_DC_U269_CLAMP.Error_T1.ATIME := T#0MS;
   S704_TL_DC_U269_CLAMP.Error_T2.IN := FALSE;
   S704_TL_DC_U269_CLAMP.Error_T2.PT := T#0MS;
   S704_TL_DC_U269_CLAMP.Error_T2.Q := FALSE;
   S704_TL_DC_U269_CLAMP.Error_T2.ET := T#0MS;
   S704_TL_DC_U269_CLAMP.Error_T2.STATE := B#16#0;
   S704_TL_DC_U269_CLAMP.Error_T2.STIME := T#0MS;
   S704_TL_DC_U269_CLAMP.Error_T2.ATIME := T#0MS;
   S704_TL_DC_U269_CLAMP.Adv_End_Aux := FALSE;
   S704_TL_DC_U269_CLAMP.Ret_End_Aux := FALSE;
   S704_TL_DC_U269_CLAMP.CHK_Aux1 := FALSE;
   S704_TL_DC_U269_CLAMP.CHK_Aux2 := FALSE;
   S704_TL_DC_U269_CLAMP.Error_T1_DN := FALSE;
   S704_TL_DC_U269_CLAMP.Error_T2_DN := FALSE;
   S704_TL_DC_U269_CLAMP.Adv_Memo := FALSE;
   S704_TL_DC_U269_CLAMP.Visu_Adv_Arr[0] := FALSE;
   S704_TL_DC_U269_CLAMP.Visu_Adv_Arr[1] := FALSE;
   S704_TL_DC_U269_CLAMP.Visu_Adv_Arr[2] := FALSE;
   S704_TL_DC_U269_CLAMP.Visu_Adv_Arr[3] := FALSE;
   S704_TL_DC_U269_CLAMP.Visu_Adv_Arr[4] := FALSE;
   S704_TL_DC_U269_CLAMP.Visu_Adv_Arr[5] := FALSE;
   S704_TL_DC_U269_CLAMP.Visu_Adv_Arr[6] := FALSE;
   S704_TL_DC_U269_CLAMP.Visu_Adv_Arr[7] := FALSE;
   S704_TL_DC_U269_CLAMP.Visu_Adv_Arr[8] := FALSE;
   S704_TL_DC_U269_CLAMP.Visu_Adv_Arr[9] := FALSE;
   S704_TL_DC_U269_CLAMP.Visu_Adv_Arr[10] := FALSE;
   S704_TL_DC_U269_CLAMP.Visu_Adv_Arr[11] := FALSE;
   S704_TL_DC_U269_CLAMP.Visu_Adv_Arr[12] := FALSE;
   S704_TL_DC_U269_CLAMP.Visu_Adv_Arr[13] := FALSE;
   S704_TL_DC_U269_CLAMP.Visu_Adv_Arr[14] := FALSE;
   S704_TL_DC_U269_CLAMP.Visu_Adv_Arr[15] := FALSE;
   S704_TL_DC_U269_CLAMP.Visu_Ret_Arr[0] := FALSE;
   S704_TL_DC_U269_CLAMP.Visu_Ret_Arr[1] := FALSE;
   S704_TL_DC_U269_CLAMP.Visu_Ret_Arr[2] := FALSE;
   S704_TL_DC_U269_CLAMP.Visu_Ret_Arr[3] := FALSE;
   S704_TL_DC_U269_CLAMP.Visu_Ret_Arr[4] := FALSE;
   S704_TL_DC_U269_CLAMP.Visu_Ret_Arr[5] := FALSE;
   S704_TL_DC_U269_CLAMP.Visu_Ret_Arr[6] := FALSE;
   S704_TL_DC_U269_CLAMP.Visu_Ret_Arr[7] := FALSE;
   S704_TL_DC_U269_CLAMP.Visu_Ret_Arr[8] := FALSE;
   S704_TL_DC_U269_CLAMP.Visu_Ret_Arr[9] := FALSE;
   S704_TL_DC_U269_CLAMP.Visu_Ret_Arr[10] := FALSE;
   S704_TL_DC_U269_CLAMP.Visu_Ret_Arr[11] := FALSE;
   S704_TL_DC_U269_CLAMP.Visu_Ret_Arr[12] := FALSE;
   S704_TL_DC_U269_CLAMP.Visu_Ret_Arr[13] := FALSE;
   S704_TL_DC_U269_CLAMP.Visu_Ret_Arr[14] := FALSE;
   S704_TL_DC_U269_CLAMP.Visu_Ret_Arr[15] := FALSE;
   S704_TL_DC_U269_CLAMP.BLK_Move_Ret := 0;
   S704_TL_DC_U269_CLAMP.Enable := FALSE;
   S704_TL_DC_U269_CLAMP.Adv_End := FALSE;
   S704_TL_DC_U269_CLAMP.Ret_End := FALSE;
   S704_TL_DC_3RD_CLAMP.Enable_Aux := FALSE;
   S704_TL_DC_3RD_CLAMP.Adv_Amount := 0;
   S704_TL_DC_3RD_CLAMP.Ret_Amount := 0;
   S704_TL_DC_3RD_CLAMP.LS_Adv1 := FALSE;
   S704_TL_DC_3RD_CLAMP.LS_Ret1 := FALSE;
   S704_TL_DC_3RD_CLAMP.LS_Adv2 := FALSE;
   S704_TL_DC_3RD_CLAMP.LS_Ret2 := FALSE;
   S704_TL_DC_3RD_CLAMP.LS_Adv3 := FALSE;
   S704_TL_DC_3RD_CLAMP.LS_Ret3 := FALSE;
   S704_TL_DC_3RD_CLAMP.LS_Adv4 := FALSE;
   S704_TL_DC_3RD_CLAMP.LS_Ret4 := FALSE;
   S704_TL_DC_3RD_CLAMP.LS_Adv5 := FALSE;
   S704_TL_DC_3RD_CLAMP.LS_Ret5 := FALSE;
   S704_TL_DC_3RD_CLAMP.LS_Adv6 := FALSE;
   S704_TL_DC_3RD_CLAMP.LS_Ret6 := FALSE;
   S704_TL_DC_3RD_CLAMP.LS_Adv7 := FALSE;
   S704_TL_DC_3RD_CLAMP.LS_Ret7 := FALSE;
   S704_TL_DC_3RD_CLAMP.LS_Adv8 := FALSE;
   S704_TL_DC_3RD_CLAMP.LS_Ret8 := FALSE;
   S704_TL_DC_3RD_CLAMP.SOL_Adv := FALSE;
   S704_TL_DC_3RD_CLAMP.SOL_Ret := FALSE;
   S704_TL_DC_3RD_CLAMP.M_Ready := FALSE;
   S704_TL_DC_3RD_CLAMP.T_CHK1 := T#0MS;
   S704_TL_DC_3RD_CLAMP.T_CHK2 := T#0MS;
   S704_TL_DC_3RD_CLAMP.PB_Lamp_CHK := FALSE;
   S704_TL_DC_3RD_CLAMP.PB_Error_Rst := FALSE;
   S704_TL_DC_3RD_CLAMP.M_FLICK := FALSE;
   S704_TL_DC_3RD_CLAMP.M_Adv_Err := FALSE;
   S704_TL_DC_3RD_CLAMP.M_Ret_Err := FALSE;
   S704_TL_DC_3RD_CLAMP.LP_Adv := FALSE;
   S704_TL_DC_3RD_CLAMP.LP_Ret := FALSE;
   S704_TL_DC_3RD_CLAMP.Visu_Adv := W#16#0;
   S704_TL_DC_3RD_CLAMP.Visu_Ret := W#16#0;
   S704_TL_DC_3RD_CLAMP.Error_T1.IN := FALSE;
   S704_TL_DC_3RD_CLAMP.Error_T1.PT := T#0MS;
   S704_TL_DC_3RD_CLAMP.Error_T1.Q := FALSE;
   S704_TL_DC_3RD_CLAMP.Error_T1.ET := T#0MS;
   S704_TL_DC_3RD_CLAMP.Error_T1.STATE := B#16#0;
   S704_TL_DC_3RD_CLAMP.Error_T1.STIME := T#0MS;
   S704_TL_DC_3RD_CLAMP.Error_T1.ATIME := T#0MS;
   S704_TL_DC_3RD_CLAMP.Error_T2.IN := FALSE;
   S704_TL_DC_3RD_CLAMP.Error_T2.PT := T#0MS;
   S704_TL_DC_3RD_CLAMP.Error_T2.Q := FALSE;
   S704_TL_DC_3RD_CLAMP.Error_T2.ET := T#0MS;
   S704_TL_DC_3RD_CLAMP.Error_T2.STATE := B#16#0;
   S704_TL_DC_3RD_CLAMP.Error_T2.STIME := T#0MS;
   S704_TL_DC_3RD_CLAMP.Error_T2.ATIME := T#0MS;
   S704_TL_DC_3RD_CLAMP.Adv_End_Aux := FALSE;
   S704_TL_DC_3RD_CLAMP.Ret_End_Aux := FALSE;
   S704_TL_DC_3RD_CLAMP.CHK_Aux1 := FALSE;
   S704_TL_DC_3RD_CLAMP.CHK_Aux2 := FALSE;
   S704_TL_DC_3RD_CLAMP.Error_T1_DN := FALSE;
   S704_TL_DC_3RD_CLAMP.Error_T2_DN := FALSE;
   S704_TL_DC_3RD_CLAMP.Adv_Memo := FALSE;
   S704_TL_DC_3RD_CLAMP.Visu_Adv_Arr[0] := FALSE;
   S704_TL_DC_3RD_CLAMP.Visu_Adv_Arr[1] := FALSE;
   S704_TL_DC_3RD_CLAMP.Visu_Adv_Arr[2] := FALSE;
   S704_TL_DC_3RD_CLAMP.Visu_Adv_Arr[3] := FALSE;
   S704_TL_DC_3RD_CLAMP.Visu_Adv_Arr[4] := FALSE;
   S704_TL_DC_3RD_CLAMP.Visu_Adv_Arr[5] := FALSE;
   S704_TL_DC_3RD_CLAMP.Visu_Adv_Arr[6] := FALSE;
   S704_TL_DC_3RD_CLAMP.Visu_Adv_Arr[7] := FALSE;
   S704_TL_DC_3RD_CLAMP.Visu_Adv_Arr[8] := FALSE;
   S704_TL_DC_3RD_CLAMP.Visu_Adv_Arr[9] := FALSE;
   S704_TL_DC_3RD_CLAMP.Visu_Adv_Arr[10] := FALSE;
   S704_TL_DC_3RD_CLAMP.Visu_Adv_Arr[11] := FALSE;
   S704_TL_DC_3RD_CLAMP.Visu_Adv_Arr[12] := FALSE;
   S704_TL_DC_3RD_CLAMP.Visu_Adv_Arr[13] := FALSE;
   S704_TL_DC_3RD_CLAMP.Visu_Adv_Arr[14] := FALSE;
   S704_TL_DC_3RD_CLAMP.Visu_Adv_Arr[15] := FALSE;
   S704_TL_DC_3RD_CLAMP.Visu_Ret_Arr[0] := FALSE;
   S704_TL_DC_3RD_CLAMP.Visu_Ret_Arr[1] := FALSE;
   S704_TL_DC_3RD_CLAMP.Visu_Ret_Arr[2] := FALSE;
   S704_TL_DC_3RD_CLAMP.Visu_Ret_Arr[3] := FALSE;
   S704_TL_DC_3RD_CLAMP.Visu_Ret_Arr[4] := FALSE;
   S704_TL_DC_3RD_CLAMP.Visu_Ret_Arr[5] := FALSE;
   S704_TL_DC_3RD_CLAMP.Visu_Ret_Arr[6] := FALSE;
   S704_TL_DC_3RD_CLAMP.Visu_Ret_Arr[7] := FALSE;
   S704_TL_DC_3RD_CLAMP.Visu_Ret_Arr[8] := FALSE;
   S704_TL_DC_3RD_CLAMP.Visu_Ret_Arr[9] := FALSE;
   S704_TL_DC_3RD_CLAMP.Visu_Ret_Arr[10] := FALSE;
   S704_TL_DC_3RD_CLAMP.Visu_Ret_Arr[11] := FALSE;
   S704_TL_DC_3RD_CLAMP.Visu_Ret_Arr[12] := FALSE;
   S704_TL_DC_3RD_CLAMP.Visu_Ret_Arr[13] := FALSE;
   S704_TL_DC_3RD_CLAMP.Visu_Ret_Arr[14] := FALSE;
   S704_TL_DC_3RD_CLAMP.Visu_Ret_Arr[15] := FALSE;
   S704_TL_DC_3RD_CLAMP.BLK_Move_Ret := 0;
   S704_TL_DC_3RD_CLAMP.Enable := FALSE;
   S704_TL_DC_3RD_CLAMP.Adv_End := FALSE;
   S704_TL_DC_3RD_CLAMP.Ret_End := FALSE;
   S704_TL_DC_U262_1_UP_DN.Enable_Aux := FALSE;
   S704_TL_DC_U262_1_UP_DN.Adv_Amount := 0;
   S704_TL_DC_U262_1_UP_DN.Ret_Amount := 0;
   S704_TL_DC_U262_1_UP_DN.LS_Adv1 := FALSE;
   S704_TL_DC_U262_1_UP_DN.LS_Ret1 := FALSE;
   S704_TL_DC_U262_1_UP_DN.LS_Adv2 := FALSE;
   S704_TL_DC_U262_1_UP_DN.LS_Ret2 := FALSE;
   S704_TL_DC_U262_1_UP_DN.LS_Adv3 := FALSE;
   S704_TL_DC_U262_1_UP_DN.LS_Ret3 := FALSE;
   S704_TL_DC_U262_1_UP_DN.LS_Adv4 := FALSE;
   S704_TL_DC_U262_1_UP_DN.LS_Ret4 := FALSE;
   S704_TL_DC_U262_1_UP_DN.LS_Adv5 := FALSE;
   S704_TL_DC_U262_1_UP_DN.LS_Ret5 := FALSE;
   S704_TL_DC_U262_1_UP_DN.LS_Adv6 := FALSE;
   S704_TL_DC_U262_1_UP_DN.LS_Ret6 := FALSE;
   S704_TL_DC_U262_1_UP_DN.LS_Adv7 := FALSE;
   S704_TL_DC_U262_1_UP_DN.LS_Ret7 := FALSE;
   S704_TL_DC_U262_1_UP_DN.LS_Adv8 := FALSE;
   S704_TL_DC_U262_1_UP_DN.LS_Ret8 := FALSE;
   S704_TL_DC_U262_1_UP_DN.SOL_Adv := FALSE;
   S704_TL_DC_U262_1_UP_DN.SOL_Ret := FALSE;
   S704_TL_DC_U262_1_UP_DN.M_Ready := FALSE;
   S704_TL_DC_U262_1_UP_DN.T_CHK1 := T#0MS;
   S704_TL_DC_U262_1_UP_DN.T_CHK2 := T#0MS;
   S704_TL_DC_U262_1_UP_DN.PB_Lamp_CHK := FALSE;
   S704_TL_DC_U262_1_UP_DN.PB_Error_Rst := FALSE;
   S704_TL_DC_U262_1_UP_DN.M_FLICK := FALSE;
   S704_TL_DC_U262_1_UP_DN.M_Adv_Err := FALSE;
   S704_TL_DC_U262_1_UP_DN.M_Ret_Err := FALSE;
   S704_TL_DC_U262_1_UP_DN.LP_Adv := FALSE;
   S704_TL_DC_U262_1_UP_DN.LP_Ret := FALSE;
   S704_TL_DC_U262_1_UP_DN.Visu_Adv := W#16#0;
   S704_TL_DC_U262_1_UP_DN.Visu_Ret := W#16#0;
   S704_TL_DC_U262_1_UP_DN.Error_T1.IN := FALSE;
   S704_TL_DC_U262_1_UP_DN.Error_T1.PT := T#0MS;
   S704_TL_DC_U262_1_UP_DN.Error_T1.Q := FALSE;
   S704_TL_DC_U262_1_UP_DN.Error_T1.ET := T#0MS;
   S704_TL_DC_U262_1_UP_DN.Error_T1.STATE := B#16#0;
   S704_TL_DC_U262_1_UP_DN.Error_T1.STIME := T#0MS;
   S704_TL_DC_U262_1_UP_DN.Error_T1.ATIME := T#0MS;
   S704_TL_DC_U262_1_UP_DN.Error_T2.IN := FALSE;
   S704_TL_DC_U262_1_UP_DN.Error_T2.PT := T#0MS;
   S704_TL_DC_U262_1_UP_DN.Error_T2.Q := FALSE;
   S704_TL_DC_U262_1_UP_DN.Error_T2.ET := T#0MS;
   S704_TL_DC_U262_1_UP_DN.Error_T2.STATE := B#16#0;
   S704_TL_DC_U262_1_UP_DN.Error_T2.STIME := T#0MS;
   S704_TL_DC_U262_1_UP_DN.Error_T2.ATIME := T#0MS;
   S704_TL_DC_U262_1_UP_DN.Adv_End_Aux := FALSE;
   S704_TL_DC_U262_1_UP_DN.Ret_End_Aux := FALSE;
   S704_TL_DC_U262_1_UP_DN.CHK_Aux1 := FALSE;
   S704_TL_DC_U262_1_UP_DN.CHK_Aux2 := FALSE;
   S704_TL_DC_U262_1_UP_DN.Error_T1_DN := FALSE;
   S704_TL_DC_U262_1_UP_DN.Error_T2_DN := FALSE;
   S704_TL_DC_U262_1_UP_DN.Adv_Memo := FALSE;
   S704_TL_DC_U262_1_UP_DN.Visu_Adv_Arr[0] := FALSE;
   S704_TL_DC_U262_1_UP_DN.Visu_Adv_Arr[1] := FALSE;
   S704_TL_DC_U262_1_UP_DN.Visu_Adv_Arr[2] := FALSE;
   S704_TL_DC_U262_1_UP_DN.Visu_Adv_Arr[3] := FALSE;
   S704_TL_DC_U262_1_UP_DN.Visu_Adv_Arr[4] := FALSE;
   S704_TL_DC_U262_1_UP_DN.Visu_Adv_Arr[5] := FALSE;
   S704_TL_DC_U262_1_UP_DN.Visu_Adv_Arr[6] := FALSE;
   S704_TL_DC_U262_1_UP_DN.Visu_Adv_Arr[7] := FALSE;
   S704_TL_DC_U262_1_UP_DN.Visu_Adv_Arr[8] := FALSE;
   S704_TL_DC_U262_1_UP_DN.Visu_Adv_Arr[9] := FALSE;
   S704_TL_DC_U262_1_UP_DN.Visu_Adv_Arr[10] := FALSE;
   S704_TL_DC_U262_1_UP_DN.Visu_Adv_Arr[11] := FALSE;
   S704_TL_DC_U262_1_UP_DN.Visu_Adv_Arr[12] := FALSE;
   S704_TL_DC_U262_1_UP_DN.Visu_Adv_Arr[13] := FALSE;
   S704_TL_DC_U262_1_UP_DN.Visu_Adv_Arr[14] := FALSE;
   S704_TL_DC_U262_1_UP_DN.Visu_Adv_Arr[15] := FALSE;
   S704_TL_DC_U262_1_UP_DN.Visu_Ret_Arr[0] := FALSE;
   S704_TL_DC_U262_1_UP_DN.Visu_Ret_Arr[1] := FALSE;
   S704_TL_DC_U262_1_UP_DN.Visu_Ret_Arr[2] := FALSE;
   S704_TL_DC_U262_1_UP_DN.Visu_Ret_Arr[3] := FALSE;
   S704_TL_DC_U262_1_UP_DN.Visu_Ret_Arr[4] := FALSE;
   S704_TL_DC_U262_1_UP_DN.Visu_Ret_Arr[5] := FALSE;
   S704_TL_DC_U262_1_UP_DN.Visu_Ret_Arr[6] := FALSE;
   S704_TL_DC_U262_1_UP_DN.Visu_Ret_Arr[7] := FALSE;
   S704_TL_DC_U262_1_UP_DN.Visu_Ret_Arr[8] := FALSE;
   S704_TL_DC_U262_1_UP_DN.Visu_Ret_Arr[9] := FALSE;
   S704_TL_DC_U262_1_UP_DN.Visu_Ret_Arr[10] := FALSE;
   S704_TL_DC_U262_1_UP_DN.Visu_Ret_Arr[11] := FALSE;
   S704_TL_DC_U262_1_UP_DN.Visu_Ret_Arr[12] := FALSE;
   S704_TL_DC_U262_1_UP_DN.Visu_Ret_Arr[13] := FALSE;
   S704_TL_DC_U262_1_UP_DN.Visu_Ret_Arr[14] := FALSE;
   S704_TL_DC_U262_1_UP_DN.Visu_Ret_Arr[15] := FALSE;
   S704_TL_DC_U262_1_UP_DN.BLK_Move_Ret := 0;
   S704_TL_DC_U262_1_UP_DN.Enable := FALSE;
   S704_TL_DC_U262_1_UP_DN.Adv_End := FALSE;
   S704_TL_DC_U262_1_UP_DN.Ret_End := FALSE;
   S704_TL_DC_U262_1.Enable_Aux := FALSE;
   S704_TL_DC_U262_1.Adv_Amount := 0;
   S704_TL_DC_U262_1.Ret_Amount := 0;
   S704_TL_DC_U262_1.LS_Adv1 := FALSE;
   S704_TL_DC_U262_1.LS_Ret1 := FALSE;
   S704_TL_DC_U262_1.LS_Adv2 := FALSE;
   S704_TL_DC_U262_1.LS_Ret2 := FALSE;
   S704_TL_DC_U262_1.LS_Adv3 := FALSE;
   S704_TL_DC_U262_1.LS_Ret3 := FALSE;
   S704_TL_DC_U262_1.LS_Adv4 := FALSE;
   S704_TL_DC_U262_1.LS_Ret4 := FALSE;
   S704_TL_DC_U262_1.LS_Adv5 := FALSE;
   S704_TL_DC_U262_1.LS_Ret5 := FALSE;
   S704_TL_DC_U262_1.LS_Adv6 := FALSE;
   S704_TL_DC_U262_1.LS_Ret6 := FALSE;
   S704_TL_DC_U262_1.LS_Adv7 := FALSE;
   S704_TL_DC_U262_1.LS_Ret7 := FALSE;
   S704_TL_DC_U262_1.LS_Adv8 := FALSE;
   S704_TL_DC_U262_1.LS_Ret8 := FALSE;
   S704_TL_DC_U262_1.SOL_Adv := FALSE;
   S704_TL_DC_U262_1.SOL_Ret := FALSE;
   S704_TL_DC_U262_1.M_Ready := FALSE;
   S704_TL_DC_U262_1.T_CHK1 := T#0MS;
   S704_TL_DC_U262_1.T_CHK2 := T#0MS;
   S704_TL_DC_U262_1.PB_Lamp_CHK := FALSE;
   S704_TL_DC_U262_1.PB_Error_Rst := FALSE;
   S704_TL_DC_U262_1.M_FLICK := FALSE;
   S704_TL_DC_U262_1.M_Adv_Err := FALSE;
   S704_TL_DC_U262_1.M_Ret_Err := FALSE;
   S704_TL_DC_U262_1.LP_Adv := FALSE;
   S704_TL_DC_U262_1.LP_Ret := FALSE;
   S704_TL_DC_U262_1.Visu_Adv := W#16#0;
   S704_TL_DC_U262_1.Visu_Ret := W#16#0;
   S704_TL_DC_U262_1.Error_T1.IN := FALSE;
   S704_TL_DC_U262_1.Error_T1.PT := T#0MS;
   S704_TL_DC_U262_1.Error_T1.Q := FALSE;
   S704_TL_DC_U262_1.Error_T1.ET := T#0MS;
   S704_TL_DC_U262_1.Error_T1.STATE := B#16#0;
   S704_TL_DC_U262_1.Error_T1.STIME := T#0MS;
   S704_TL_DC_U262_1.Error_T1.ATIME := T#0MS;
   S704_TL_DC_U262_1.Error_T2.IN := FALSE;
   S704_TL_DC_U262_1.Error_T2.PT := T#0MS;
   S704_TL_DC_U262_1.Error_T2.Q := FALSE;
   S704_TL_DC_U262_1.Error_T2.ET := T#0MS;
   S704_TL_DC_U262_1.Error_T2.STATE := B#16#0;
   S704_TL_DC_U262_1.Error_T2.STIME := T#0MS;
   S704_TL_DC_U262_1.Error_T2.ATIME := T#0MS;
   S704_TL_DC_U262_1.Adv_End_Aux := FALSE;
   S704_TL_DC_U262_1.Ret_End_Aux := FALSE;
   S704_TL_DC_U262_1.CHK_Aux1 := FALSE;
   S704_TL_DC_U262_1.CHK_Aux2 := FALSE;
   S704_TL_DC_U262_1.Error_T1_DN := FALSE;
   S704_TL_DC_U262_1.Error_T2_DN := FALSE;
   S704_TL_DC_U262_1.Adv_Memo := FALSE;
   S704_TL_DC_U262_1.Visu_Adv_Arr[0] := FALSE;
   S704_TL_DC_U262_1.Visu_Adv_Arr[1] := FALSE;
   S704_TL_DC_U262_1.Visu_Adv_Arr[2] := FALSE;
   S704_TL_DC_U262_1.Visu_Adv_Arr[3] := FALSE;
   S704_TL_DC_U262_1.Visu_Adv_Arr[4] := FALSE;
   S704_TL_DC_U262_1.Visu_Adv_Arr[5] := FALSE;
   S704_TL_DC_U262_1.Visu_Adv_Arr[6] := FALSE;
   S704_TL_DC_U262_1.Visu_Adv_Arr[7] := FALSE;
   S704_TL_DC_U262_1.Visu_Adv_Arr[8] := FALSE;
   S704_TL_DC_U262_1.Visu_Adv_Arr[9] := FALSE;
   S704_TL_DC_U262_1.Visu_Adv_Arr[10] := FALSE;
   S704_TL_DC_U262_1.Visu_Adv_Arr[11] := FALSE;
   S704_TL_DC_U262_1.Visu_Adv_Arr[12] := FALSE;
   S704_TL_DC_U262_1.Visu_Adv_Arr[13] := FALSE;
   S704_TL_DC_U262_1.Visu_Adv_Arr[14] := FALSE;
   S704_TL_DC_U262_1.Visu_Adv_Arr[15] := FALSE;
   S704_TL_DC_U262_1.Visu_Ret_Arr[0] := FALSE;
   S704_TL_DC_U262_1.Visu_Ret_Arr[1] := FALSE;
   S704_TL_DC_U262_1.Visu_Ret_Arr[2] := FALSE;
   S704_TL_DC_U262_1.Visu_Ret_Arr[3] := FALSE;
   S704_TL_DC_U262_1.Visu_Ret_Arr[4] := FALSE;
   S704_TL_DC_U262_1.Visu_Ret_Arr[5] := FALSE;
   S704_TL_DC_U262_1.Visu_Ret_Arr[6] := FALSE;
   S704_TL_DC_U262_1.Visu_Ret_Arr[7] := FALSE;
   S704_TL_DC_U262_1.Visu_Ret_Arr[8] := FALSE;
   S704_TL_DC_U262_1.Visu_Ret_Arr[9] := FALSE;
   S704_TL_DC_U262_1.Visu_Ret_Arr[10] := FALSE;
   S704_TL_DC_U262_1.Visu_Ret_Arr[11] := FALSE;
   S704_TL_DC_U262_1.Visu_Ret_Arr[12] := FALSE;
   S704_TL_DC_U262_1.Visu_Ret_Arr[13] := FALSE;
   S704_TL_DC_U262_1.Visu_Ret_Arr[14] := FALSE;
   S704_TL_DC_U262_1.Visu_Ret_Arr[15] := FALSE;
   S704_TL_DC_U262_1.BLK_Move_Ret := 0;
   S704_TL_DC_U262_1.Enable := FALSE;
   S704_TL_DC_U262_1.Adv_End := FALSE;
   S704_TL_DC_U262_1.Ret_End := FALSE;
   S704_TL_DC_U262_1_CLAMP.Enable_Aux := FALSE;
   S704_TL_DC_U262_1_CLAMP.Adv_Amount := 0;
   S704_TL_DC_U262_1_CLAMP.Ret_Amount := 0;
   S704_TL_DC_U262_1_CLAMP.LS_Adv1 := FALSE;
   S704_TL_DC_U262_1_CLAMP.LS_Ret1 := FALSE;
   S704_TL_DC_U262_1_CLAMP.LS_Adv2 := FALSE;
   S704_TL_DC_U262_1_CLAMP.LS_Ret2 := FALSE;
   S704_TL_DC_U262_1_CLAMP.LS_Adv3 := FALSE;
   S704_TL_DC_U262_1_CLAMP.LS_Ret3 := FALSE;
   S704_TL_DC_U262_1_CLAMP.LS_Adv4 := FALSE;
   S704_TL_DC_U262_1_CLAMP.LS_Ret4 := FALSE;
   S704_TL_DC_U262_1_CLAMP.LS_Adv5 := FALSE;
   S704_TL_DC_U262_1_CLAMP.LS_Ret5 := FALSE;
   S704_TL_DC_U262_1_CLAMP.LS_Adv6 := FALSE;
   S704_TL_DC_U262_1_CLAMP.LS_Ret6 := FALSE;
   S704_TL_DC_U262_1_CLAMP.LS_Adv7 := FALSE;
   S704_TL_DC_U262_1_CLAMP.LS_Ret7 := FALSE;
   S704_TL_DC_U262_1_CLAMP.LS_Adv8 := FALSE;
   S704_TL_DC_U262_1_CLAMP.LS_Ret8 := FALSE;
   S704_TL_DC_U262_1_CLAMP.SOL_Adv := FALSE;
   S704_TL_DC_U262_1_CLAMP.SOL_Ret := FALSE;
   S704_TL_DC_U262_1_CLAMP.M_Ready := FALSE;
   S704_TL_DC_U262_1_CLAMP.T_CHK1 := T#0MS;
   S704_TL_DC_U262_1_CLAMP.T_CHK2 := T#0MS;
   S704_TL_DC_U262_1_CLAMP.PB_Lamp_CHK := FALSE;
   S704_TL_DC_U262_1_CLAMP.PB_Error_Rst := FALSE;
   S704_TL_DC_U262_1_CLAMP.M_FLICK := FALSE;
   S704_TL_DC_U262_1_CLAMP.M_Adv_Err := FALSE;
   S704_TL_DC_U262_1_CLAMP.M_Ret_Err := FALSE;
   S704_TL_DC_U262_1_CLAMP.LP_Adv := FALSE;
   S704_TL_DC_U262_1_CLAMP.LP_Ret := FALSE;
   S704_TL_DC_U262_1_CLAMP.Visu_Adv := W#16#0;
   S704_TL_DC_U262_1_CLAMP.Visu_Ret := W#16#0;
   S704_TL_DC_U262_1_CLAMP.Error_T1.IN := FALSE;
   S704_TL_DC_U262_1_CLAMP.Error_T1.PT := T#0MS;
   S704_TL_DC_U262_1_CLAMP.Error_T1.Q := FALSE;
   S704_TL_DC_U262_1_CLAMP.Error_T1.ET := T#0MS;
   S704_TL_DC_U262_1_CLAMP.Error_T1.STATE := B#16#0;
   S704_TL_DC_U262_1_CLAMP.Error_T1.STIME := T#0MS;
   S704_TL_DC_U262_1_CLAMP.Error_T1.ATIME := T#0MS;
   S704_TL_DC_U262_1_CLAMP.Error_T2.IN := FALSE;
   S704_TL_DC_U262_1_CLAMP.Error_T2.PT := T#0MS;
   S704_TL_DC_U262_1_CLAMP.Error_T2.Q := FALSE;
   S704_TL_DC_U262_1_CLAMP.Error_T2.ET := T#0MS;
   S704_TL_DC_U262_1_CLAMP.Error_T2.STATE := B#16#0;
   S704_TL_DC_U262_1_CLAMP.Error_T2.STIME := T#0MS;
   S704_TL_DC_U262_1_CLAMP.Error_T2.ATIME := T#0MS;
   S704_TL_DC_U262_1_CLAMP.Adv_End_Aux := FALSE;
   S704_TL_DC_U262_1_CLAMP.Ret_End_Aux := FALSE;
   S704_TL_DC_U262_1_CLAMP.CHK_Aux1 := FALSE;
   S704_TL_DC_U262_1_CLAMP.CHK_Aux2 := FALSE;
   S704_TL_DC_U262_1_CLAMP.Error_T1_DN := FALSE;
   S704_TL_DC_U262_1_CLAMP.Error_T2_DN := FALSE;
   S704_TL_DC_U262_1_CLAMP.Adv_Memo := FALSE;
   S704_TL_DC_U262_1_CLAMP.Visu_Adv_Arr[0] := FALSE;
   S704_TL_DC_U262_1_CLAMP.Visu_Adv_Arr[1] := FALSE;
   S704_TL_DC_U262_1_CLAMP.Visu_Adv_Arr[2] := FALSE;
   S704_TL_DC_U262_1_CLAMP.Visu_Adv_Arr[3] := FALSE;
   S704_TL_DC_U262_1_CLAMP.Visu_Adv_Arr[4] := FALSE;
   S704_TL_DC_U262_1_CLAMP.Visu_Adv_Arr[5] := FALSE;
   S704_TL_DC_U262_1_CLAMP.Visu_Adv_Arr[6] := FALSE;
   S704_TL_DC_U262_1_CLAMP.Visu_Adv_Arr[7] := FALSE;
   S704_TL_DC_U262_1_CLAMP.Visu_Adv_Arr[8] := FALSE;
   S704_TL_DC_U262_1_CLAMP.Visu_Adv_Arr[9] := FALSE;
   S704_TL_DC_U262_1_CLAMP.Visu_Adv_Arr[10] := FALSE;
   S704_TL_DC_U262_1_CLAMP.Visu_Adv_Arr[11] := FALSE;
   S704_TL_DC_U262_1_CLAMP.Visu_Adv_Arr[12] := FALSE;
   S704_TL_DC_U262_1_CLAMP.Visu_Adv_Arr[13] := FALSE;
   S704_TL_DC_U262_1_CLAMP.Visu_Adv_Arr[14] := FALSE;
   S704_TL_DC_U262_1_CLAMP.Visu_Adv_Arr[15] := FALSE;
   S704_TL_DC_U262_1_CLAMP.Visu_Ret_Arr[0] := FALSE;
   S704_TL_DC_U262_1_CLAMP.Visu_Ret_Arr[1] := FALSE;
   S704_TL_DC_U262_1_CLAMP.Visu_Ret_Arr[2] := FALSE;
   S704_TL_DC_U262_1_CLAMP.Visu_Ret_Arr[3] := FALSE;
   S704_TL_DC_U262_1_CLAMP.Visu_Ret_Arr[4] := FALSE;
   S704_TL_DC_U262_1_CLAMP.Visu_Ret_Arr[5] := FALSE;
   S704_TL_DC_U262_1_CLAMP.Visu_Ret_Arr[6] := FALSE;
   S704_TL_DC_U262_1_CLAMP.Visu_Ret_Arr[7] := FALSE;
   S704_TL_DC_U262_1_CLAMP.Visu_Ret_Arr[8] := FALSE;
   S704_TL_DC_U262_1_CLAMP.Visu_Ret_Arr[9] := FALSE;
   S704_TL_DC_U262_1_CLAMP.Visu_Ret_Arr[10] := FALSE;
   S704_TL_DC_U262_1_CLAMP.Visu_Ret_Arr[11] := FALSE;
   S704_TL_DC_U262_1_CLAMP.Visu_Ret_Arr[12] := FALSE;
   S704_TL_DC_U262_1_CLAMP.Visu_Ret_Arr[13] := FALSE;
   S704_TL_DC_U262_1_CLAMP.Visu_Ret_Arr[14] := FALSE;
   S704_TL_DC_U262_1_CLAMP.Visu_Ret_Arr[15] := FALSE;
   S704_TL_DC_U262_1_CLAMP.BLK_Move_Ret := 0;
   S704_TL_DC_U262_1_CLAMP.Enable := FALSE;
   S704_TL_DC_U262_1_CLAMP.Adv_End := FALSE;
   S704_TL_DC_U262_1_CLAMP.Ret_End := FALSE;
   S704_TL_DC_U261_2_CLAMP.Enable_Aux := FALSE;
   S704_TL_DC_U261_2_CLAMP.Adv_Amount := 0;
   S704_TL_DC_U261_2_CLAMP.Ret_Amount := 0;
   S704_TL_DC_U261_2_CLAMP.LS_Adv1 := FALSE;
   S704_TL_DC_U261_2_CLAMP.LS_Ret1 := FALSE;
   S704_TL_DC_U261_2_CLAMP.LS_Adv2 := FALSE;
   S704_TL_DC_U261_2_CLAMP.LS_Ret2 := FALSE;
   S704_TL_DC_U261_2_CLAMP.LS_Adv3 := FALSE;
   S704_TL_DC_U261_2_CLAMP.LS_Ret3 := FALSE;
   S704_TL_DC_U261_2_CLAMP.LS_Adv4 := FALSE;
   S704_TL_DC_U261_2_CLAMP.LS_Ret4 := FALSE;
   S704_TL_DC_U261_2_CLAMP.LS_Adv5 := FALSE;
   S704_TL_DC_U261_2_CLAMP.LS_Ret5 := FALSE;
   S704_TL_DC_U261_2_CLAMP.LS_Adv6 := FALSE;
   S704_TL_DC_U261_2_CLAMP.LS_Ret6 := FALSE;
   S704_TL_DC_U261_2_CLAMP.LS_Adv7 := FALSE;
   S704_TL_DC_U261_2_CLAMP.LS_Ret7 := FALSE;
   S704_TL_DC_U261_2_CLAMP.LS_Adv8 := FALSE;
   S704_TL_DC_U261_2_CLAMP.LS_Ret8 := FALSE;
   S704_TL_DC_U261_2_CLAMP.SOL_Adv := FALSE;
   S704_TL_DC_U261_2_CLAMP.SOL_Ret := FALSE;
   S704_TL_DC_U261_2_CLAMP.M_Ready := FALSE;
   S704_TL_DC_U261_2_CLAMP.T_CHK1 := T#0MS;
   S704_TL_DC_U261_2_CLAMP.T_CHK2 := T#0MS;
   S704_TL_DC_U261_2_CLAMP.PB_Lamp_CHK := FALSE;
   S704_TL_DC_U261_2_CLAMP.PB_Error_Rst := FALSE;
   S704_TL_DC_U261_2_CLAMP.M_FLICK := FALSE;
   S704_TL_DC_U261_2_CLAMP.M_Adv_Err := FALSE;
   S704_TL_DC_U261_2_CLAMP.M_Ret_Err := FALSE;
   S704_TL_DC_U261_2_CLAMP.LP_Adv := FALSE;
   S704_TL_DC_U261_2_CLAMP.LP_Ret := FALSE;
   S704_TL_DC_U261_2_CLAMP.Visu_Adv := W#16#0;
   S704_TL_DC_U261_2_CLAMP.Visu_Ret := W#16#0;
   S704_TL_DC_U261_2_CLAMP.Error_T1.IN := FALSE;
   S704_TL_DC_U261_2_CLAMP.Error_T1.PT := T#0MS;
   S704_TL_DC_U261_2_CLAMP.Error_T1.Q := FALSE;
   S704_TL_DC_U261_2_CLAMP.Error_T1.ET := T#0MS;
   S704_TL_DC_U261_2_CLAMP.Error_T1.STATE := B#16#0;
   S704_TL_DC_U261_2_CLAMP.Error_T1.STIME := T#0MS;
   S704_TL_DC_U261_2_CLAMP.Error_T1.ATIME := T#0MS;
   S704_TL_DC_U261_2_CLAMP.Error_T2.IN := FALSE;
   S704_TL_DC_U261_2_CLAMP.Error_T2.PT := T#0MS;
   S704_TL_DC_U261_2_CLAMP.Error_T2.Q := FALSE;
   S704_TL_DC_U261_2_CLAMP.Error_T2.ET := T#0MS;
   S704_TL_DC_U261_2_CLAMP.Error_T2.STATE := B#16#0;
   S704_TL_DC_U261_2_CLAMP.Error_T2.STIME := T#0MS;
   S704_TL_DC_U261_2_CLAMP.Error_T2.ATIME := T#0MS;
   S704_TL_DC_U261_2_CLAMP.Adv_End_Aux := FALSE;
   S704_TL_DC_U261_2_CLAMP.Ret_End_Aux := FALSE;
   S704_TL_DC_U261_2_CLAMP.CHK_Aux1 := FALSE;
   S704_TL_DC_U261_2_CLAMP.CHK_Aux2 := FALSE;
   S704_TL_DC_U261_2_CLAMP.Error_T1_DN := FALSE;
   S704_TL_DC_U261_2_CLAMP.Error_T2_DN := FALSE;
   S704_TL_DC_U261_2_CLAMP.Adv_Memo := FALSE;
   S704_TL_DC_U261_2_CLAMP.Visu_Adv_Arr[0] := FALSE;
   S704_TL_DC_U261_2_CLAMP.Visu_Adv_Arr[1] := FALSE;
   S704_TL_DC_U261_2_CLAMP.Visu_Adv_Arr[2] := FALSE;
   S704_TL_DC_U261_2_CLAMP.Visu_Adv_Arr[3] := FALSE;
   S704_TL_DC_U261_2_CLAMP.Visu_Adv_Arr[4] := FALSE;
   S704_TL_DC_U261_2_CLAMP.Visu_Adv_Arr[5] := FALSE;
   S704_TL_DC_U261_2_CLAMP.Visu_Adv_Arr[6] := FALSE;
   S704_TL_DC_U261_2_CLAMP.Visu_Adv_Arr[7] := FALSE;
   S704_TL_DC_U261_2_CLAMP.Visu_Adv_Arr[8] := FALSE;
   S704_TL_DC_U261_2_CLAMP.Visu_Adv_Arr[9] := FALSE;
   S704_TL_DC_U261_2_CLAMP.Visu_Adv_Arr[10] := FALSE;
   S704_TL_DC_U261_2_CLAMP.Visu_Adv_Arr[11] := FALSE;
   S704_TL_DC_U261_2_CLAMP.Visu_Adv_Arr[12] := FALSE;
   S704_TL_DC_U261_2_CLAMP.Visu_Adv_Arr[13] := FALSE;
   S704_TL_DC_U261_2_CLAMP.Visu_Adv_Arr[14] := FALSE;
   S704_TL_DC_U261_2_CLAMP.Visu_Adv_Arr[15] := FALSE;
   S704_TL_DC_U261_2_CLAMP.Visu_Ret_Arr[0] := FALSE;
   S704_TL_DC_U261_2_CLAMP.Visu_Ret_Arr[1] := FALSE;
   S704_TL_DC_U261_2_CLAMP.Visu_Ret_Arr[2] := FALSE;
   S704_TL_DC_U261_2_CLAMP.Visu_Ret_Arr[3] := FALSE;
   S704_TL_DC_U261_2_CLAMP.Visu_Ret_Arr[4] := FALSE;
   S704_TL_DC_U261_2_CLAMP.Visu_Ret_Arr[5] := FALSE;
   S704_TL_DC_U261_2_CLAMP.Visu_Ret_Arr[6] := FALSE;
   S704_TL_DC_U261_2_CLAMP.Visu_Ret_Arr[7] := FALSE;
   S704_TL_DC_U261_2_CLAMP.Visu_Ret_Arr[8] := FALSE;
   S704_TL_DC_U261_2_CLAMP.Visu_Ret_Arr[9] := FALSE;
   S704_TL_DC_U261_2_CLAMP.Visu_Ret_Arr[10] := FALSE;
   S704_TL_DC_U261_2_CLAMP.Visu_Ret_Arr[11] := FALSE;
   S704_TL_DC_U261_2_CLAMP.Visu_Ret_Arr[12] := FALSE;
   S704_TL_DC_U261_2_CLAMP.Visu_Ret_Arr[13] := FALSE;
   S704_TL_DC_U261_2_CLAMP.Visu_Ret_Arr[14] := FALSE;
   S704_TL_DC_U261_2_CLAMP.Visu_Ret_Arr[15] := FALSE;
   S704_TL_DC_U261_2_CLAMP.BLK_Move_Ret := 0;
   S704_TL_DC_U261_2_CLAMP.Enable := FALSE;
   S704_TL_DC_U261_2_CLAMP.Adv_End := FALSE;
   S704_TL_DC_U261_2_CLAMP.Ret_End := FALSE;
END_DATA_BLOCK

FUNCTION FC 144 : VOID
TITLE =
VERSION : 0.1

BEGIN
NETWORK
TITLE =
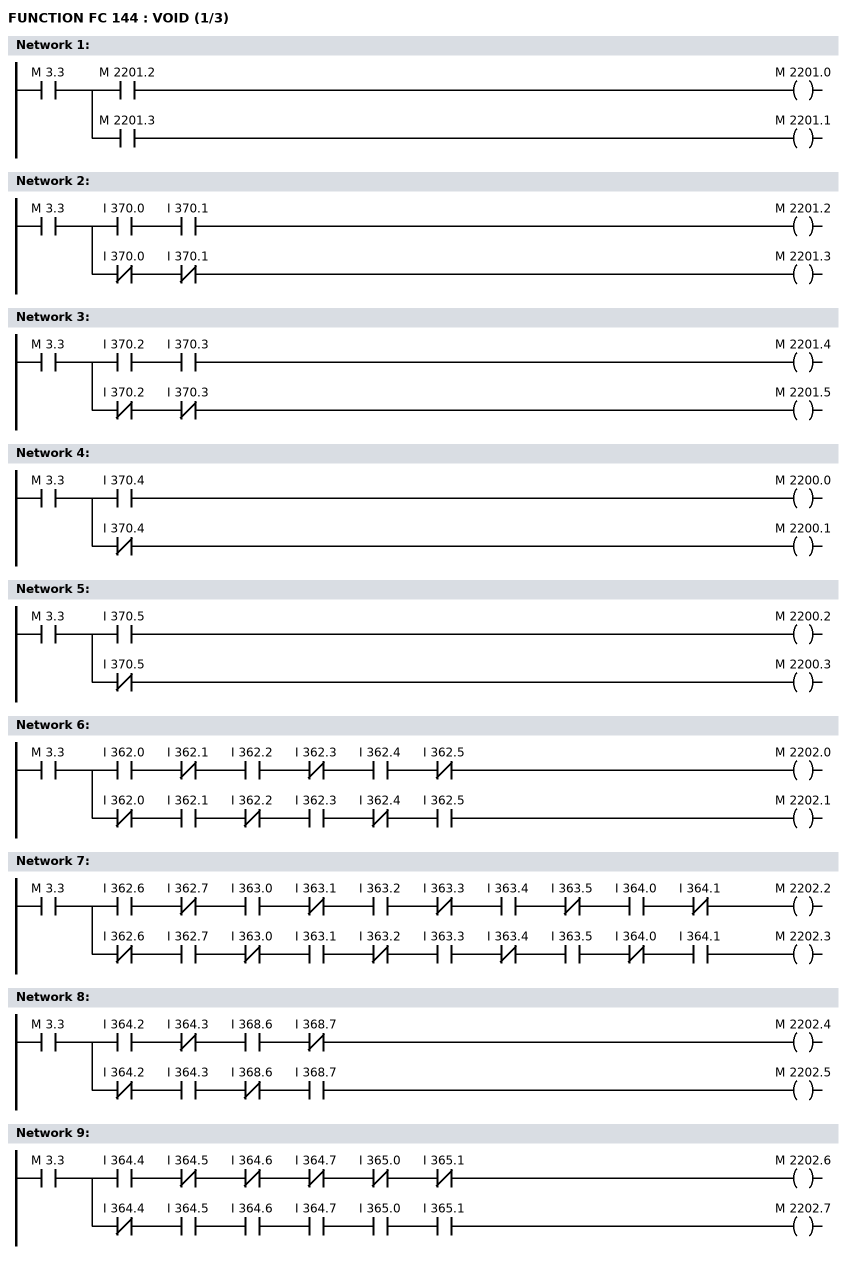

      A     M      3.3;
      =     L      0.0;
      A     L      0.0;
      A     M   2201.2;
      =     M   2201.0;
      A     L      0.0;
      A     M   2201.3;
      =     M   2201.1;
NETWORK
TITLE =

      A     M      3.3;
      =     L      0.0;
      A     L      0.0;
      A     I    370.0;
      A     I    370.1;
      =     M   2201.2;
      A     L      0.0;
      AN    I    370.0;
      AN    I    370.1;
      =     M   2201.3;
NETWORK
TITLE =

      A     M      3.3;
      =     L      0.0;
      A     L      0.0;
      A     I    370.2;
      A     I    370.3;
      =     M   2201.4;
      A     L      0.0;
      AN    I    370.2;
      AN    I    370.3;
      =     M   2201.5;
NETWORK
TITLE =

      A     M      3.3;
      =     L      0.0;
      A     L      0.0;
      A     I    370.4;
      =     M   2200.0;
      A     L      0.0;
      AN    I    370.4;
      =     M   2200.1;
NETWORK
TITLE =

      A     M      3.3;
      =     L      0.0;
      A     L      0.0;
      A     I    370.5;
      =     M   2200.2;
      A     L      0.0;
      AN    I    370.5;
      =     M   2200.3;
NETWORK
TITLE =

      A     M      3.3;
      =     L      0.0;
      A     L      0.0;
      A     I    362.0;
      AN    I    362.1;
      A     I    362.2;
      AN    I    362.3;
      A     I    362.4;
      AN    I    362.5;
      =     M   2202.0;
      A     L      0.0;
      AN    I    362.0;
      A     I    362.1;
      AN    I    362.2;
      A     I    362.3;
      AN    I    362.4;
      A     I    362.5;
      =     M   2202.1;
NETWORK
TITLE =

      A     M      3.3;
      =     L      0.0;
      A     L      0.0;
      A     I    362.6;
      AN    I    362.7;
      A     I    363.0;
      AN    I    363.1;
      A     I    363.2;
      AN    I    363.3;
      A     I    363.4;
      AN    I    363.5;
      A     I    364.0;
      AN    I    364.1;
      =     M   2202.2;
      A     L      0.0;
      AN    I    362.6;
      A     I    362.7;
      AN    I    363.0;
      A     I    363.1;
      AN    I    363.2;
      A     I    363.3;
      AN    I    363.4;
      A     I    363.5;
      AN    I    364.0;
      A     I    364.1;
      =     M   2202.3;
NETWORK
TITLE =

      A     M      3.3;
      =     L      0.0;
      A     L      0.0;
      A     I    364.2;
      AN    I    364.3;
      A     I    368.6;
      AN    I    368.7;
      =     M   2202.4;
      A     L      0.0;
      AN    I    364.2;
      A     I    364.3;
      AN    I    368.6;
      A     I    368.7;
      =     M   2202.5;
NETWORK
TITLE =

      A     M      3.3;
      =     L      0.0;
      A     L      0.0;
      A     I    364.4;
      AN    I    364.5;
      AN    I    364.6;
      AN    I    364.7;
      AN    I    365.0;
      AN    I    365.1;
      =     M   2202.6;
      A     L      0.0;
      AN    I    364.4;
      A     I    364.5;
      A     I    364.6;
      A     I    364.7;
      A     I    365.0;
      A     I    365.1;
      =     M   2202.7;
NETWORK
TITLE =
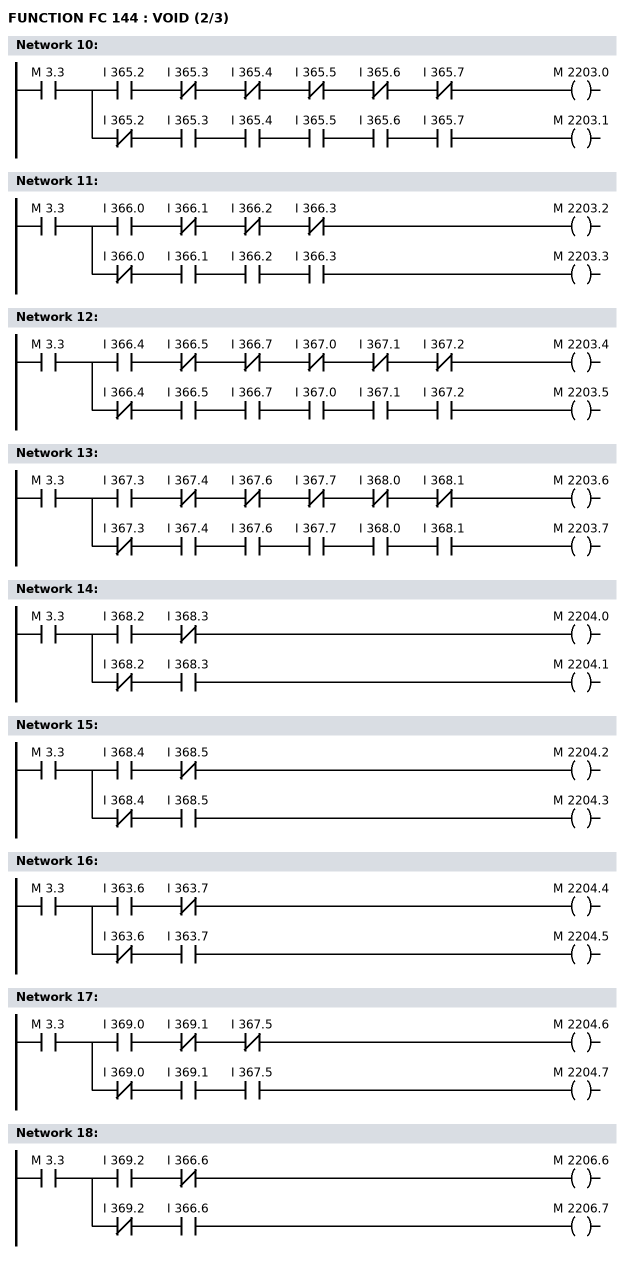

      A     M      3.3;
      =     L      0.0;
      A     L      0.0;
      A     I    365.2;
      AN    I    365.3;
      AN    I    365.4;
      AN    I    365.5;
      AN    I    365.6;
      AN    I    365.7;
      =     M   2203.0;
      A     L      0.0;
      AN    I    365.2;
      A     I    365.3;
      A     I    365.4;
      A     I    365.5;
      A     I    365.6;
      A     I    365.7;
      =     M   2203.1;
NETWORK
TITLE =

      A     M      3.3;
      =     L      0.0;
      A     L      0.0;
      A     I    366.0;
      AN    I    366.1;
      AN    I    366.2;
      AN    I    366.3;
      =     M   2203.2;
      A     L      0.0;
      AN    I    366.0;
      A     I    366.1;
      A     I    366.2;
      A     I    366.3;
      =     M   2203.3;
NETWORK
TITLE =

      A     M      3.3;
      =     L      0.0;
      A     L      0.0;
      A     I    366.4;
      AN    I    366.5;
      AN    I    366.7;
      AN    I    367.0;
      AN    I    367.1;
      AN    I    367.2;
      =     M   2203.4;
      A     L      0.0;
      AN    I    366.4;
      A     I    366.5;
      A     I    366.7;
      A     I    367.0;
      A     I    367.1;
      A     I    367.2;
      =     M   2203.5;
NETWORK
TITLE =

      A     M      3.3;
      =     L      0.0;
      A     L      0.0;
      A     I    367.3;
      AN    I    367.4;
      AN    I    367.6;
      AN    I    367.7;
      AN    I    368.0;
      AN    I    368.1;
      =     M   2203.6;
      A     L      0.0;
      AN    I    367.3;
      A     I    367.4;
      A     I    367.6;
      A     I    367.7;
      A     I    368.0;
      A     I    368.1;
      =     M   2203.7;
NETWORK
TITLE =

      A     M      3.3;
      =     L      0.0;
      A     L      0.0;
      A     I    368.2;
      AN    I    368.3;
      =     M   2204.0;
      A     L      0.0;
      AN    I    368.2;
      A     I    368.3;
      =     M   2204.1;
NETWORK
TITLE =

      A     M      3.3;
      =     L      0.0;
      A     L      0.0;
      A     I    368.4;
      AN    I    368.5;
      =     M   2204.2;
      A     L      0.0;
      AN    I    368.4;
      A     I    368.5;
      =     M   2204.3;
NETWORK
TITLE =

      A     M      3.3;
      =     L      0.0;
      A     L      0.0;
      A     I    363.6;
      AN    I    363.7;
      =     M   2204.4;
      A     L      0.0;
      AN    I    363.6;
      A     I    363.7;
      =     M   2204.5;
NETWORK
TITLE =

      A     M      3.3;
      =     L      0.0;
      A     L      0.0;
      A     I    369.0;
      AN    I    369.1;
      AN    I    367.5;
      =     M   2204.6;
      A     L      0.0;
      AN    I    369.0;
      A     I    369.1;
      A     I    367.5;
      =     M   2204.7;
NETWORK
TITLE =

      A     M      3.3;
      =     L      0.0;
      A     L      0.0;
      A     I    369.2;
      AN    I    366.6;
      =     M   2206.6;
      A     L      0.0;
      AN    I    369.2;
      A     I    366.6;
      =     M   2206.7;
NETWORK
TITLE =
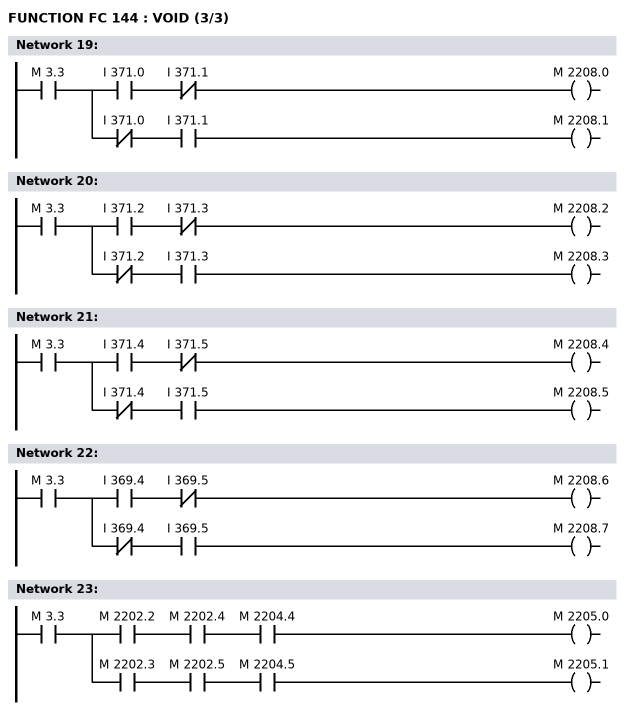

      A     M      3.3;
      =     L      0.0;
      A     L      0.0;
      A     I    371.0;
      AN    I    371.1;
      =     M   2208.0;
      A     L      0.0;
      AN    I    371.0;
      A     I    371.1;
      =     M   2208.1;
NETWORK
TITLE =

      A     M      3.3;
      =     L      0.0;
      A     L      0.0;
      A     I    371.2;
      AN    I    371.3;
      =     M   2208.2;
      A     L      0.0;
      AN    I    371.2;
      A     I    371.3;
      =     M   2208.3;
NETWORK
TITLE =

      A     M      3.3;
      =     L      0.0;
      A     L      0.0;
      A     I    371.4;
      AN    I    371.5;
      =     M   2208.4;
      A     L      0.0;
      AN    I    371.4;
      A     I    371.5;
      =     M   2208.5;
NETWORK
TITLE =

      A     M      3.3;
      =     L      0.0;
      A     L      0.0;
      A     I    369.4;
      AN    I    369.5;
      =     M   2208.6;
      A     L      0.0;
      AN    I    369.4;
      A     I    369.5;
      =     M   2208.7;
NETWORK
TITLE =

      A     M      3.3;
      =     L      0.0;
      A     L      0.0;
      A     M   2202.2;
      A     M   2202.4;
      A     M   2204.4;
      =     M   2205.0;
      A     L      0.0;
      A     M   2202.3;
      A     M   2202.5;
      A     M   2204.5;
      =     M   2205.1;
NETWORK
TITLE =

      A     M      3.3;
      =     L      0.0;
      A     L      0.0;
      A     M   2202.6;
      A     M   2203.0;
      A     M   2203.2;
      A     M   2203.4;
      A     M   2203.6;
      A     M   2206.6;
      =     L      0.1;
      A     L      0.1;
      BLD   102;
      =     M   2205.2;
      A     L      0.1;
      A     M   2204.2;
      A     M   2204.6;
      =     M   2205.4;
      A     L      0.0;
      A     M   2202.7;
      A     M   2203.1;
      A     M   2203.3;
      A     M   2203.5;
      A     M   2203.7;
      A     M   2206.7;
      =     L      0.1;
      A     L      0.1;
      BLD   102;
      =     M   2205.3;
      A     L      0.1;
      A     M   2204.3;
      A     M   2204.7;
      =     M   2205.5;
NETWORK
TITLE =
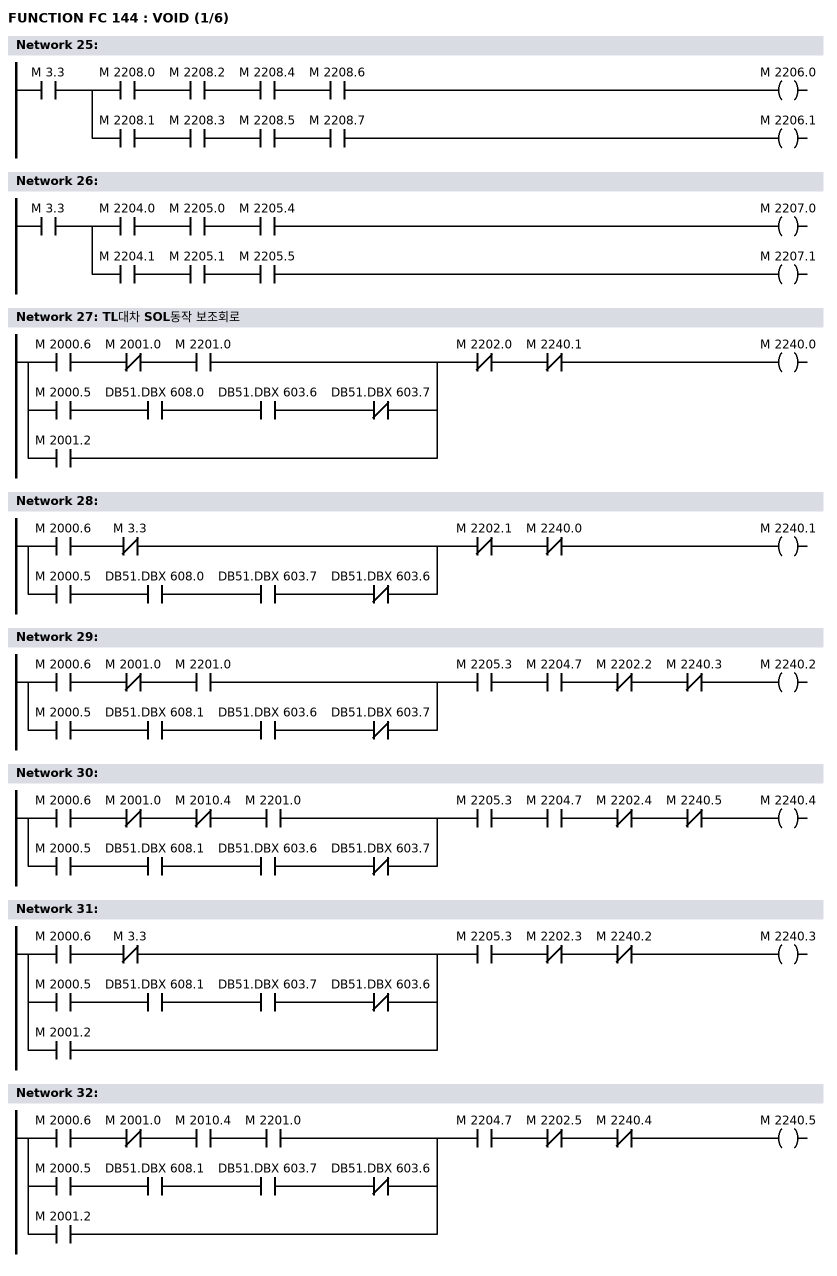

      A     M      3.3;
      =     L      0.0;
      A     L      0.0;
      A     M   2208.0;
      A     M   2208.2;
      A     M   2208.4;
      A     M   2208.6;
      =     M   2206.0;
      A     L      0.0;
      A     M   2208.1;
      A     M   2208.3;
      A     M   2208.5;
      A     M   2208.7;
      =     M   2206.1;
NETWORK
TITLE =

      A     M      3.3;
      =     L      0.0;
      A     L      0.0;
      A     M   2204.0;
      A     M   2205.0;
      A     M   2205.4;
      =     M   2207.0;
      A     L      0.0;
      A     M   2204.1;
      A     M   2205.1;
      A     M   2205.5;
      =     M   2207.1;
NETWORK
TITLE =TL대차 SOL동작 보조회로

      A(    ;
      A     M   2000.6;
      AN    M   2001.0;
      A     M   2201.0;
      O     ;
      A     M   2000.5;
      A     DB51.DBX  608.0;
      A     DB51.DBX  603.6;
      AN    DB51.DBX  603.7;
      O     M   2001.2;
      )     ;
      AN    M   2202.0;
      AN    M   2240.1;
      =     M   2240.0;
NETWORK
TITLE =

      A(    ;
      A     M   2000.6;
      AN    M      3.3;
      O     ;
      A     M   2000.5;
      A     DB51.DBX  608.0;
      A     DB51.DBX  603.7;
      AN    DB51.DBX  603.6;
      )     ;
      AN    M   2202.1;
      AN    M   2240.0;
      =     M   2240.1;
NETWORK
TITLE =

      A(    ;
      A     M   2000.6;
      AN    M   2001.0;
      A     M   2201.0;
      O     ;
      A     M   2000.5;
      A     DB51.DBX  608.1;
      A     DB51.DBX  603.6;
      AN    DB51.DBX  603.7;
      )     ;
      A     M   2205.3;
      A     M   2204.7;
      AN    M   2202.2;
      AN    M   2240.3;
      =     M   2240.2;
NETWORK
TITLE =

      A(    ;
      A     M   2000.6;
      AN    M   2001.0;
      AN    M   2010.4;
      A     M   2201.0;
      O     ;
      A     M   2000.5;
      A     DB51.DBX  608.1;
      A     DB51.DBX  603.6;
      AN    DB51.DBX  603.7;
      )     ;
      A     M   2205.3;
      A     M   2204.7;
      AN    M   2202.4;
      AN    M   2240.5;
      =     M   2240.4;
NETWORK
TITLE =

      A(    ;
      A     M   2000.6;
      AN    M      3.3;
      O     ;
      A     M   2000.5;
      A     DB51.DBX  608.1;
      A     DB51.DBX  603.7;
      AN    DB51.DBX  603.6;
      O     M   2001.2;
      )     ;
      A     M   2205.3;
      AN    M   2202.3;
      AN    M   2240.2;
      =     M   2240.3;
NETWORK
TITLE =

      A(    ;
      A     M   2000.6;
      AN    M   2001.0;
      A     M   2010.4;
      A     M   2201.0;
      O     ;
      A     M   2000.5;
      A     DB51.DBX  608.1;
      A     DB51.DBX  603.7;
      AN    DB51.DBX  603.6;
      O     M   2001.2;
      )     ;
      A     M   2204.7;
      AN    M   2202.5;
      AN    M   2240.4;
      =     M   2240.5;
NETWORK
TITLE =
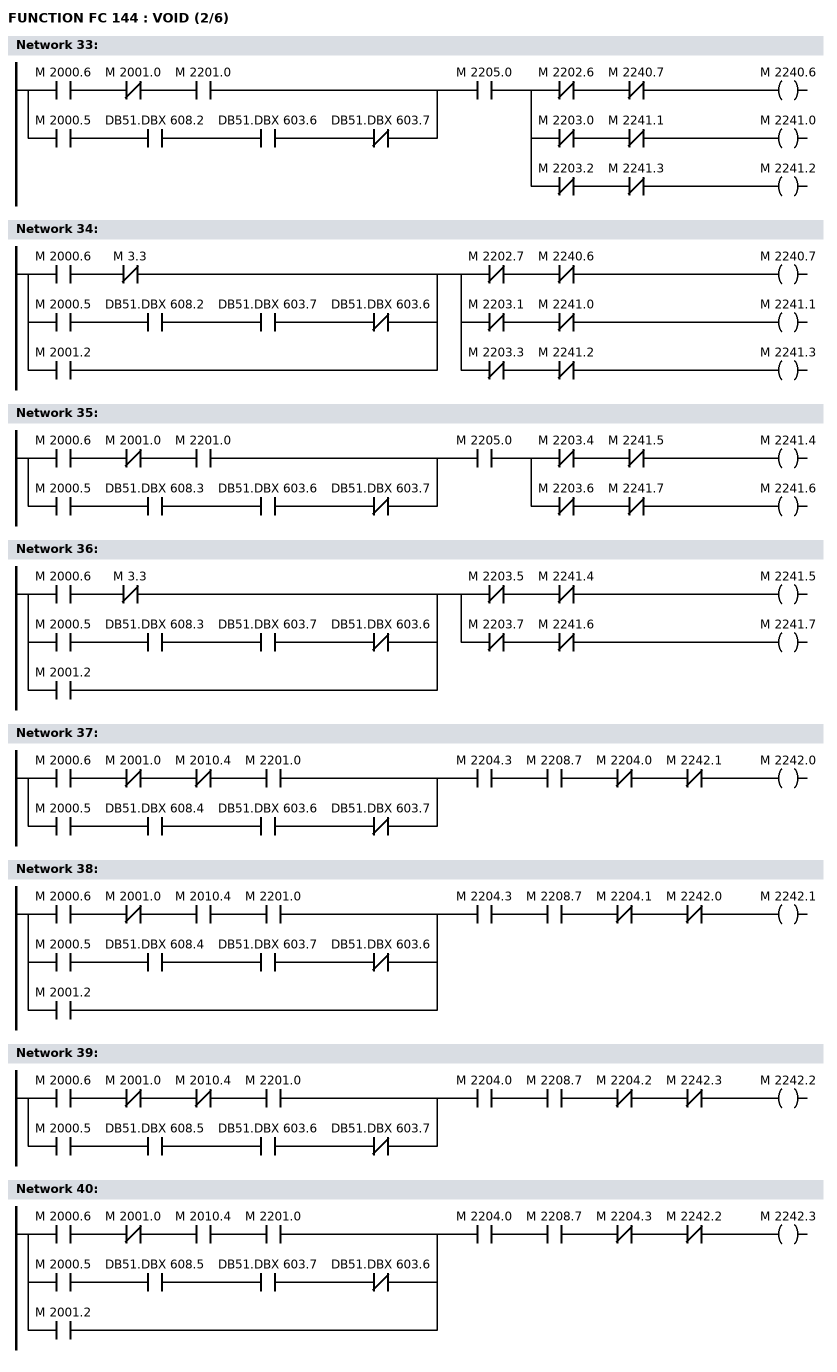

      A(    ;
      A     M   2000.6;
      AN    M   2001.0;
      A     M   2201.0;
      O     ;
      A     M   2000.5;
      A     DB51.DBX  608.2;
      A     DB51.DBX  603.6;
      AN    DB51.DBX  603.7;
      )     ;
      A     M   2205.0;
      =     L      0.0;
      A     L      0.0;
      AN    M   2202.6;
      AN    M   2240.7;
      =     M   2240.6;
      A     L      0.0;
      AN    M   2203.0;
      AN    M   2241.1;
      =     M   2241.0;
      A     L      0.0;
      AN    M   2203.2;
      AN    M   2241.3;
      =     M   2241.2;
NETWORK
TITLE =

      A     M   2000.6;
      AN    M      3.3;
      O     ;
      A     M   2000.5;
      A     DB51.DBX  608.2;
      A     DB51.DBX  603.7;
      AN    DB51.DBX  603.6;
      O     M   2001.2;
      =     L      0.0;
      A     L      0.0;
      AN    M   2202.7;
      AN    M   2240.6;
      =     M   2240.7;
      A     L      0.0;
      AN    M   2203.1;
      AN    M   2241.0;
      =     M   2241.1;
      A     L      0.0;
      AN    M   2203.3;
      AN    M   2241.2;
      =     M   2241.3;
NETWORK
TITLE =

      A(    ;
      A     M   2000.6;
      AN    M   2001.0;
      A     M   2201.0;
      O     ;
      A     M   2000.5;
      A     DB51.DBX  608.3;
      A     DB51.DBX  603.6;
      AN    DB51.DBX  603.7;
      )     ;
      A     M   2205.0;
      =     L      0.0;
      A     L      0.0;
      AN    M   2203.4;
      AN    M   2241.5;
      =     M   2241.4;
      A     L      0.0;
      AN    M   2203.6;
      AN    M   2241.7;
      =     M   2241.6;
NETWORK
TITLE =

      A     M   2000.6;
      AN    M      3.3;
      O     ;
      A     M   2000.5;
      A     DB51.DBX  608.3;
      A     DB51.DBX  603.7;
      AN    DB51.DBX  603.6;
      O     M   2001.2;
      =     L      0.0;
      A     L      0.0;
      AN    M   2203.5;
      AN    M   2241.4;
      =     M   2241.5;
      A     L      0.0;
      AN    M   2203.7;
      AN    M   2241.6;
      =     M   2241.7;
NETWORK
TITLE =

      A(    ;
      A     M   2000.6;
      AN    M   2001.0;
      AN    M   2010.4;
      A     M   2201.0;
      O     ;
      A     M   2000.5;
      A     DB51.DBX  608.4;
      A     DB51.DBX  603.6;
      AN    DB51.DBX  603.7;
      )     ;
      A     M   2204.3;
      A     M   2208.7;
      AN    M   2204.0;
      AN    M   2242.1;
      =     M   2242.0;
NETWORK
TITLE =

